// TIA Portal V20 export
FUNCTION_BLOCK "FB_IO_Device_Functional_Test"   // FB4, LAD
{ S7_Optimized_Access := 'TRUE' }
// stored: MemoryReserve 100, SetENOAutomatically false
   VAR_INPUT
      Reset_PLC_Functional_Test : Array[0..31] of Bool;
      Status : Bool;
      Voltage_Read : UInt;
      Min_Electrical_Current : UInt;
      Max_Electrical_Current : UInt;
      Time_End_Electrical_Current_Test : Time;
      Time_Start_Visual_Test : Time;
      In_Functional_Test_Odd : "IO_Device_Functinal_Test_Odd";
      In_Functional_Test_Even : "IO_Device_Functinal_Test_Even";
   END_VAR
   VAR_OUTPUT
      Out_Test_Parameters_Odd : "IO_Device_Test_Parameters_Odd";
      Out_Test_Parameters_Even : "IO_Device_Test_Parameters_Even";
      Out_Voltage_Read : UInt;
      Comunication_Error_Panel_1 : Bool;
      Comunication_Error_Panel_2 : Bool;
      Comunication_Error_Panel_3 : Bool;
      Comunication_Error_Panel_4 : Bool;
      Comunication_Error_Panel_5 : Bool;
      Comunication_Error_Panel_6 : Bool;
      Comunication_Error_Panel_7 : Bool;
      Comunication_Error_Panel_8 : Bool;
      Comunication_Error_Panel_9 : Bool;
      Comunication_Error_Panel_10 : Bool;
      Comunication_Error_Panel_11 : Bool;
      Comunication_Error_Panel_12 : Bool;
      Comunication_Error_Panel_13 : Bool;
      Comunication_Error_Panel_14 : Bool;
      Comunication_Error_Panel_15 : Bool;
      Comunication_Error_Panel_16 : Bool;
      Comunication_Error_Panel_17 : Bool;
      Comunication_Error_Panel_18 : Bool;
      Comunication_Error_Panel_19 : Bool;
      Comunication_Error_Panel_20 : Bool;
      Comunication_Error_Panel_21 : Bool;
      Comunication_Error_Panel_22 : Bool;
      Comunication_Error_Panel_23 : Bool;
      Comunication_Error_Panel_24 : Bool;
      Comunication_Error_Panel_25 : Bool;
      Comunication_Error_Panel_26 : Bool;
      Comunication_Error_Panel_27 : Bool;
      Comunication_Error_Panel_28 : Bool;
      Comunication_Error_Panel_29 : Bool;
      Comunication_Error_Panel_30 : Bool;
   END_VAR
   VAR
      Enable_Comunication_Erro_3 : Bool;
      Enable_Comunication_Erro_4 : Bool;
      Enable_Comunication_Erro_5 : Bool;
      Enable_Comunication_Erro_6 : Bool;
      Enable_Comunication_Erro_7 : Bool;
      Enable_Comunication_Erro_8 : Bool;
      Enable_Comunication_Erro_9 : Bool;
      Enable_Comunication_Erro_10 : Bool;
      Enable_Comunication_Erro_11 : Bool;
      Enable_Comunication_Erro_12 : Bool;
      Enable_Comunication_Erro_13 : Bool;
      Enable_Comunication_Erro_14 : Bool;
      Enable_Comunication_Erro_15 : Bool;
      Enable_Comunication_Erro_16 : Bool;
      Enable_Comunication_Erro_17 : Bool;
      Enable_Comunication_Erro_18 : Bool;
      Enable_Comunication_Erro_19 : Bool;
      Enable_Comunication_Erro_20 : Bool;
      Enable_Comunication_Erro_21 : Bool;
      Enable_Comunication_Erro_22 : Bool;
      Enable_Comunication_Erro_23 : Bool;
      Enable_Comunication_Erro_24 : Bool;
      Enable_Comunication_Erro_25 : Bool;
      Enable_Comunication_Erro_26 : Bool;
      Enable_Comunication_Erro_27 : Bool;
      Enable_Comunication_Erro_28 : Bool;
      Enable_Comunication_Erro_29 : Bool;
      Enable_Comunication_Erro_30 : Bool;
      Timer_Alarme_A_1 { S7_SetPoint := 'True'} : TON_TIME;
      Timer_Alarme_B_1 { S7_SetPoint := 'True'} : TON_TIME;
      Timer_Alarme_A_2 { S7_SetPoint := 'True'} : TON_TIME;
      Timer_Alarme_B_2 { S7_SetPoint := 'True'} : TON_TIME;
      Timer_Alarme_A_3 { S7_SetPoint := 'True'} : TON_TIME;
      Timer_Alarme_B_3 { S7_SetPoint := 'True'} : TON_TIME;
      Timer_Alarme_A_4 { S7_SetPoint := 'True'} : TON_TIME;
      Timer_Alarme_B_4 { S7_SetPoint := 'True'} : TON_TIME;
      Timer_Alarme_A_5 { S7_SetPoint := 'True'} : TON_TIME;
      Timer_Alarme_B_5 { S7_SetPoint := 'True'} : TON_TIME;
      Timer_Alarme_A_6 { S7_SetPoint := 'True'} : TON_TIME;
      Timer_Alarme_B_6 { S7_SetPoint := 'True'} : TON_TIME;
      Timer_Alarme_A_7 { S7_SetPoint := 'True'} : TON_TIME;
      Timer_Alarme_B_7 { S7_SetPoint := 'True'} : TON_TIME;
      Timer_Alarme_A_8 { S7_SetPoint := 'True'} : TON_TIME;
      Timer_Alarme_B_8 { S7_SetPoint := 'True'} : TON_TIME;
      Timer_Alarme_A_9 { S7_SetPoint := 'True'} : TON_TIME;
      Timer_Alarme_B_9 { S7_SetPoint := 'True'} : TON_TIME;
      Timer_Alarme_A_10 { S7_SetPoint := 'True'} : TON_TIME;
      Timer_Alarme_B_10 { S7_SetPoint := 'True'} : TON_TIME;
      Timer_Alarme_A_11 { S7_SetPoint := 'True'} : TON_TIME;
      Timer_Alarme_B_11 { S7_SetPoint := 'True'} : TON_TIME;
      Timer_Alarme_A_12 { S7_SetPoint := 'True'} : TON_TIME;
      Timer_Alarme_B_12 { S7_SetPoint := 'True'} : TON_TIME;
      Timer_Alarme_A_13 { S7_SetPoint := 'True'} : TON_TIME;
      Timer_Alarme_B_13 { S7_SetPoint := 'True'} : TON_TIME;
      Timer_Alarme_A_14 { S7_SetPoint := 'True'} : TON_TIME;
      Timer_Alarme_B_14 { S7_SetPoint := 'True'} : TON_TIME;
      Timer_Alarme_A_15 { S7_SetPoint := 'True'} : TON_TIME;
      Timer_Alarme_B_15 { S7_SetPoint := 'True'} : TON_TIME;
      Timer_Alarme_A_16 { S7_SetPoint := 'True'} : TON_TIME;
      Timer_Alarme_B_16 { S7_SetPoint := 'True'} : TON_TIME;
      Timer_Alarme_A_17 { S7_SetPoint := 'True'} : TON_TIME;
      Timer_Alarme_B_17 { S7_SetPoint := 'True'} : TON_TIME;
      Timer_Alarme_A_18 { S7_SetPoint := 'True'} : TON_TIME;
      Timer_Alarme_B_18 { S7_SetPoint := 'True'} : TON_TIME;
      Timer_Alarme_A_19 { S7_SetPoint := 'True'} : TON_TIME;
      Timer_Alarme_B_19 { S7_SetPoint := 'True'} : TON_TIME;
      Timer_Alarme_A_20 { S7_SetPoint := 'True'} : TON_TIME;
      Timer_Alarme_B_20 { S7_SetPoint := 'True'} : TON_TIME;
      Timer_Alarme_A_21 { S7_SetPoint := 'True'} : TON_TIME;
      Timer_Alarme_B_21 { S7_SetPoint := 'True'} : TON_TIME;
      Timer_Alarme_A_22 { S7_SetPoint := 'True'} : TON_TIME;
      Timer_Alarme_B_22 { S7_SetPoint := 'True'} : TON_TIME;
      Timer_Alarme_A_23 { S7_SetPoint := 'True'} : TON_TIME;
      Timer_Alarme_B_23 { S7_SetPoint := 'True'} : TON_TIME;
      Timer_Alarme_A_24 { S7_SetPoint := 'True'} : TON_TIME;
      Timer_Alarme_B_24 { S7_SetPoint := 'True'} : TON_TIME;
      Timer_Alarme_A_25 { S7_SetPoint := 'True'} : TON_TIME;
      Timer_Alarme_B_25 { S7_SetPoint := 'True'} : TON_TIME;
      Timer_Alarme_A_26 { S7_SetPoint := 'True'} : TON_TIME;
      Timer_Alarme_B_26 { S7_SetPoint := 'True'} : TON_TIME;
      Timer_Alarme_A_27 { S7_SetPoint := 'True'} : TON_TIME;
      Timer_Alarme_B_27 { S7_SetPoint := 'True'} : TON_TIME;
      Timer_Alarme_A_28 { S7_SetPoint := 'True'} : TON_TIME;
      Timer_Alarme_B_28 { S7_SetPoint := 'True'} : TON_TIME;
      Timer_Alarme_A_29 { S7_SetPoint := 'True'} : TON_TIME;
      Timer_Alarme_B_29 { S7_SetPoint := 'True'} : TON_TIME;
      Timer_Alarme_A_30 { S7_SetPoint := 'True'} : TON_TIME;
      Timer_Alarme_B_30 { S7_SetPoint := 'True'} : TON_TIME;
   END_VAR
BEGIN

REGION Network 1
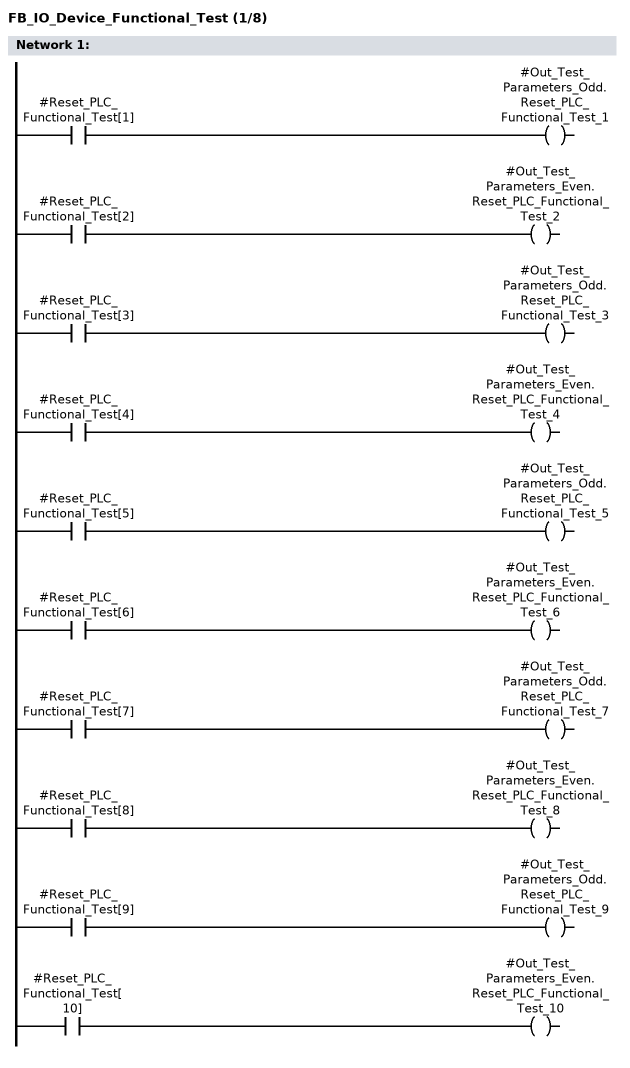
   RUNG wire#powerrail
      Contact( #Reset_PLC_Functional_Test[1] )
      Coil( #Out_Test_Parameters_Odd.Reset_PLC_Functional_Test_1 )
   END_RUNG
   RUNG wire#powerrail
      Contact( #Reset_PLC_Functional_Test[2] )
      Coil( #Out_Test_Parameters_Even.Reset_PLC_Functional_Test_2 )
   END_RUNG
   RUNG wire#powerrail
      Contact( #Reset_PLC_Functional_Test[3] )
      Coil( #Out_Test_Parameters_Odd.Reset_PLC_Functional_Test_3 )
   END_RUNG
   RUNG wire#powerrail
      Contact( #Reset_PLC_Functional_Test[4] )
      Coil( #Out_Test_Parameters_Even.Reset_PLC_Functional_Test_4 )
   END_RUNG
   RUNG wire#powerrail
      Contact( #Reset_PLC_Functional_Test[5] )
      Coil( #Out_Test_Parameters_Odd.Reset_PLC_Functional_Test_5 )
   END_RUNG
   RUNG wire#powerrail
      Contact( #Reset_PLC_Functional_Test[6] )
      Coil( #Out_Test_Parameters_Even.Reset_PLC_Functional_Test_6 )
   END_RUNG
   RUNG wire#powerrail
      Contact( #Reset_PLC_Functional_Test[7] )
      Coil( #Out_Test_Parameters_Odd.Reset_PLC_Functional_Test_7 )
   END_RUNG
   RUNG wire#powerrail
      Contact( #Reset_PLC_Functional_Test[8] )
      Coil( #Out_Test_Parameters_Even.Reset_PLC_Functional_Test_8 )
   END_RUNG
   RUNG wire#powerrail
      Contact( #Reset_PLC_Functional_Test[9] )
      Coil( #Out_Test_Parameters_Odd.Reset_PLC_Functional_Test_9 )
   END_RUNG
   RUNG wire#powerrail
      Contact( #Reset_PLC_Functional_Test[10] )
      Coil( #Out_Test_Parameters_Even.Reset_PLC_Functional_Test_10 )
   END_RUNG
   // the same network as SCL:
   #Out_Test_Parameters_Odd.Reset_PLC_Functional_Test_1 := #Reset_PLC_Functional_Test[1];
   #Out_Test_Parameters_Even.Reset_PLC_Functional_Test_2 := #Reset_PLC_Functional_Test[2];
   #Out_Test_Parameters_Odd.Reset_PLC_Functional_Test_3 := #Reset_PLC_Functional_Test[3];
   #Out_Test_Parameters_Even.Reset_PLC_Functional_Test_4 := #Reset_PLC_Functional_Test[4];
   #Out_Test_Parameters_Odd.Reset_PLC_Functional_Test_5 := #Reset_PLC_Functional_Test[5];
   #Out_Test_Parameters_Even.Reset_PLC_Functional_Test_6 := #Reset_PLC_Functional_Test[6];
   #Out_Test_Parameters_Odd.Reset_PLC_Functional_Test_7 := #Reset_PLC_Functional_Test[7];
   #Out_Test_Parameters_Even.Reset_PLC_Functional_Test_8 := #Reset_PLC_Functional_Test[8];
   #Out_Test_Parameters_Odd.Reset_PLC_Functional_Test_9 := #Reset_PLC_Functional_Test[9];
   #Out_Test_Parameters_Even.Reset_PLC_Functional_Test_10 := #Reset_PLC_Functional_Test[10];
END_REGION

REGION Network 2
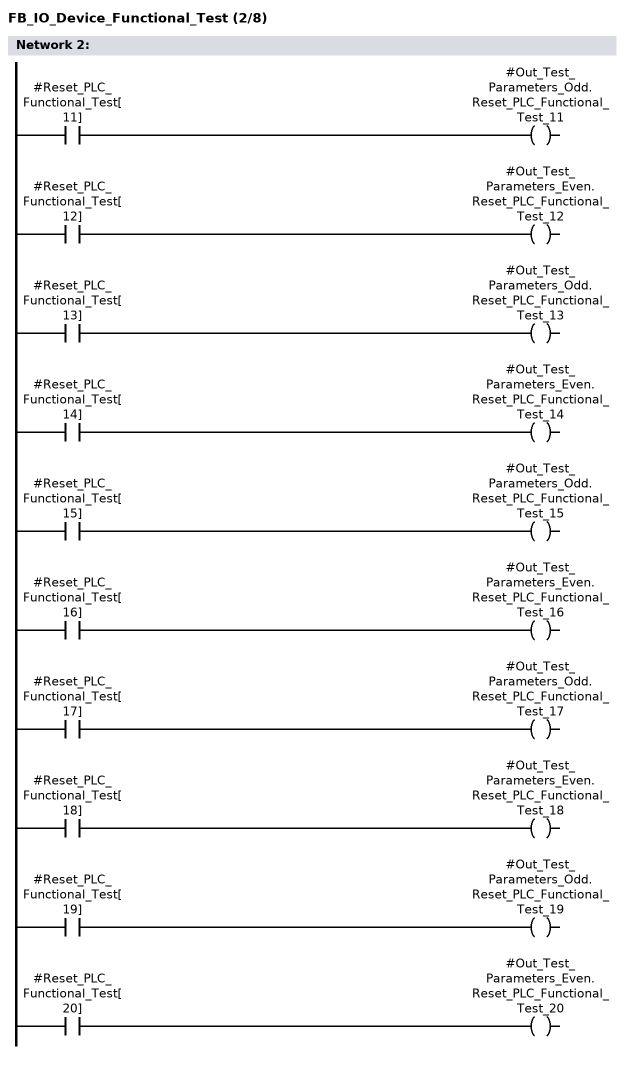
   RUNG wire#powerrail
      Contact( #Reset_PLC_Functional_Test[11] )
      Coil( #Out_Test_Parameters_Odd.Reset_PLC_Functional_Test_11 )
   END_RUNG
   RUNG wire#powerrail
      Contact( #Reset_PLC_Functional_Test[12] )
      Coil( #Out_Test_Parameters_Even.Reset_PLC_Functional_Test_12 )
   END_RUNG
   RUNG wire#powerrail
      Contact( #Reset_PLC_Functional_Test[13] )
      Coil( #Out_Test_Parameters_Odd.Reset_PLC_Functional_Test_13 )
   END_RUNG
   RUNG wire#powerrail
      Contact( #Reset_PLC_Functional_Test[14] )
      Coil( #Out_Test_Parameters_Even.Reset_PLC_Functional_Test_14 )
   END_RUNG
   RUNG wire#powerrail
      Contact( #Reset_PLC_Functional_Test[15] )
      Coil( #Out_Test_Parameters_Odd.Reset_PLC_Functional_Test_15 )
   END_RUNG
   RUNG wire#powerrail
      Contact( #Reset_PLC_Functional_Test[16] )
      Coil( #Out_Test_Parameters_Even.Reset_PLC_Functional_Test_16 )
   END_RUNG
   RUNG wire#powerrail
      Contact( #Reset_PLC_Functional_Test[17] )
      Coil( #Out_Test_Parameters_Odd.Reset_PLC_Functional_Test_17 )
   END_RUNG
   RUNG wire#powerrail
      Contact( #Reset_PLC_Functional_Test[18] )
      Coil( #Out_Test_Parameters_Even.Reset_PLC_Functional_Test_18 )
   END_RUNG
   RUNG wire#powerrail
      Contact( #Reset_PLC_Functional_Test[19] )
      Coil( #Out_Test_Parameters_Odd.Reset_PLC_Functional_Test_19 )
   END_RUNG
   RUNG wire#powerrail
      Contact( #Reset_PLC_Functional_Test[20] )
      Coil( #Out_Test_Parameters_Even.Reset_PLC_Functional_Test_20 )
   END_RUNG
   // the same network as SCL:
   #Out_Test_Parameters_Odd.Reset_PLC_Functional_Test_11 := #Reset_PLC_Functional_Test[11];
   #Out_Test_Parameters_Even.Reset_PLC_Functional_Test_12 := #Reset_PLC_Functional_Test[12];
   #Out_Test_Parameters_Odd.Reset_PLC_Functional_Test_13 := #Reset_PLC_Functional_Test[13];
   #Out_Test_Parameters_Even.Reset_PLC_Functional_Test_14 := #Reset_PLC_Functional_Test[14];
   #Out_Test_Parameters_Odd.Reset_PLC_Functional_Test_15 := #Reset_PLC_Functional_Test[15];
   #Out_Test_Parameters_Even.Reset_PLC_Functional_Test_16 := #Reset_PLC_Functional_Test[16];
   #Out_Test_Parameters_Odd.Reset_PLC_Functional_Test_17 := #Reset_PLC_Functional_Test[17];
   #Out_Test_Parameters_Even.Reset_PLC_Functional_Test_18 := #Reset_PLC_Functional_Test[18];
   #Out_Test_Parameters_Odd.Reset_PLC_Functional_Test_19 := #Reset_PLC_Functional_Test[19];
   #Out_Test_Parameters_Even.Reset_PLC_Functional_Test_20 := #Reset_PLC_Functional_Test[20];
END_REGION

REGION Network 3
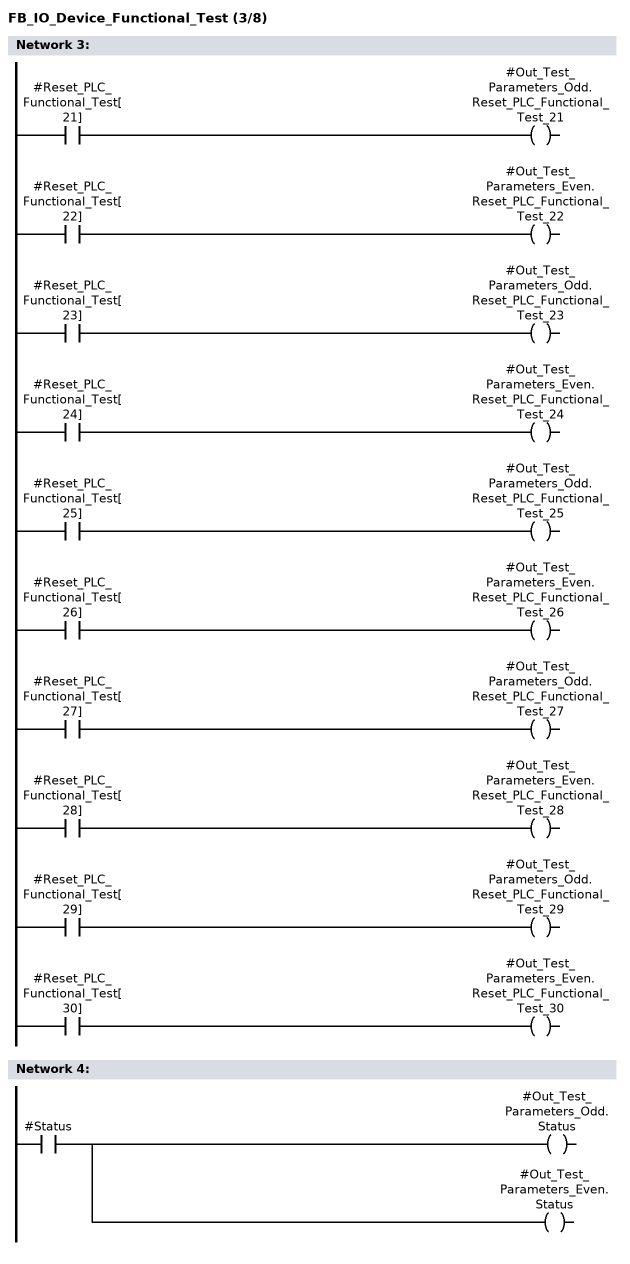
   RUNG wire#powerrail
      Contact( #Reset_PLC_Functional_Test[21] )
      Coil( #Out_Test_Parameters_Odd.Reset_PLC_Functional_Test_21 )
   END_RUNG
   RUNG wire#powerrail
      Contact( #Reset_PLC_Functional_Test[22] )
      Coil( #Out_Test_Parameters_Even.Reset_PLC_Functional_Test_22 )
   END_RUNG
   RUNG wire#powerrail
      Contact( #Reset_PLC_Functional_Test[23] )
      Coil( #Out_Test_Parameters_Odd.Reset_PLC_Functional_Test_23 )
   END_RUNG
   RUNG wire#powerrail
      Contact( #Reset_PLC_Functional_Test[24] )
      Coil( #Out_Test_Parameters_Even.Reset_PLC_Functional_Test_24 )
   END_RUNG
   RUNG wire#powerrail
      Contact( #Reset_PLC_Functional_Test[25] )
      Coil( #Out_Test_Parameters_Odd.Reset_PLC_Functional_Test_25 )
   END_RUNG
   RUNG wire#powerrail
      Contact( #Reset_PLC_Functional_Test[26] )
      Coil( #Out_Test_Parameters_Even.Reset_PLC_Functional_Test_26 )
   END_RUNG
   RUNG wire#powerrail
      Contact( #Reset_PLC_Functional_Test[27] )
      Coil( #Out_Test_Parameters_Odd.Reset_PLC_Functional_Test_27 )
   END_RUNG
   RUNG wire#powerrail
      Contact( #Reset_PLC_Functional_Test[28] )
      Coil( #Out_Test_Parameters_Even.Reset_PLC_Functional_Test_28 )
   END_RUNG
   RUNG wire#powerrail
      Contact( #Reset_PLC_Functional_Test[29] )
      Coil( #Out_Test_Parameters_Odd.Reset_PLC_Functional_Test_29 )
   END_RUNG
   RUNG wire#powerrail
      Contact( #Reset_PLC_Functional_Test[30] )
      Coil( #Out_Test_Parameters_Even.Reset_PLC_Functional_Test_30 )
   END_RUNG
   // the same network as SCL:
   #Out_Test_Parameters_Odd.Reset_PLC_Functional_Test_21 := #Reset_PLC_Functional_Test[21];
   #Out_Test_Parameters_Even.Reset_PLC_Functional_Test_22 := #Reset_PLC_Functional_Test[22];
   #Out_Test_Parameters_Odd.Reset_PLC_Functional_Test_23 := #Reset_PLC_Functional_Test[23];
   #Out_Test_Parameters_Even.Reset_PLC_Functional_Test_24 := #Reset_PLC_Functional_Test[24];
   #Out_Test_Parameters_Odd.Reset_PLC_Functional_Test_25 := #Reset_PLC_Functional_Test[25];
   #Out_Test_Parameters_Even.Reset_PLC_Functional_Test_26 := #Reset_PLC_Functional_Test[26];
   #Out_Test_Parameters_Odd.Reset_PLC_Functional_Test_27 := #Reset_PLC_Functional_Test[27];
   #Out_Test_Parameters_Even.Reset_PLC_Functional_Test_28 := #Reset_PLC_Functional_Test[28];
   #Out_Test_Parameters_Odd.Reset_PLC_Functional_Test_29 := #Reset_PLC_Functional_Test[29];
   #Out_Test_Parameters_Even.Reset_PLC_Functional_Test_30 := #Reset_PLC_Functional_Test[30];
END_REGION

REGION Network 4
   RUNG wire#powerrail
      Contact( #Status )
      wire#w1
      Coil( #Out_Test_Parameters_Odd.Status )
   END_RUNG
   RUNG wire#w1
      Coil( #Out_Test_Parameters_Even.Status )
   END_RUNG
   // the same network as SCL:
   #Out_Test_Parameters_Odd.Status := #Status;
   #Out_Test_Parameters_Even.Status := #Status;
END_REGION

REGION Network 5
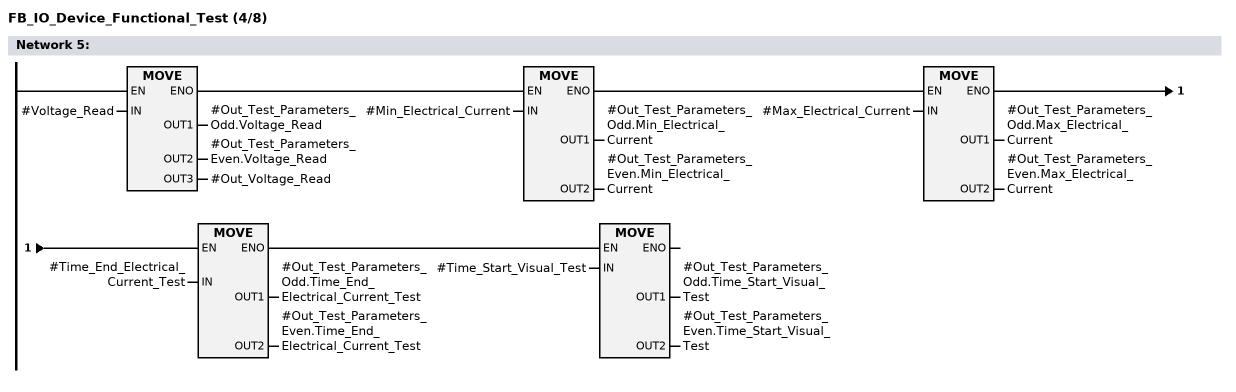
   RUNG wire#powerrail
      Move(in := #Voltage_Read, out1 => #Out_Test_Parameters_Odd.Voltage_Read, out2 => #Out_Test_Parameters_Even.Voltage_Read, out3 => #Out_Voltage_Read)
      Move(in := #Min_Electrical_Current, out1 => #Out_Test_Parameters_Odd.Min_Electrical_Current, out2 => #Out_Test_Parameters_Even.Min_Electrical_Current)
      Move(in := #Max_Electrical_Current, out1 => #Out_Test_Parameters_Odd.Max_Electrical_Current, out2 => #Out_Test_Parameters_Even.Max_Electrical_Current)
      Move(in := #Time_End_Electrical_Current_Test, out1 => #Out_Test_Parameters_Odd.Time_End_Electrical_Current_Test, out2 => #Out_Test_Parameters_Even.Time_End_Electrical_Current_Test)
      Move(in := #Time_Start_Visual_Test, out1 => #Out_Test_Parameters_Odd.Time_Start_Visual_Test, out2 => #Out_Test_Parameters_Even.Time_Start_Visual_Test)
   END_RUNG
   // the same network as SCL:
   #Out_Test_Parameters_Odd.Voltage_Read := #Voltage_Read;
   #Out_Test_Parameters_Even.Voltage_Read := #Voltage_Read;
   #Out_Voltage_Read := #Voltage_Read;
   #Out_Test_Parameters_Odd.Min_Electrical_Current := #Min_Electrical_Current;
   #Out_Test_Parameters_Even.Min_Electrical_Current := #Min_Electrical_Current;
   #Out_Test_Parameters_Odd.Max_Electrical_Current := #Max_Electrical_Current;
   #Out_Test_Parameters_Even.Max_Electrical_Current := #Max_Electrical_Current;
   #Out_Test_Parameters_Odd.Time_End_Electrical_Current_Test := #Time_End_Electrical_Current_Test;
   #Out_Test_Parameters_Even.Time_End_Electrical_Current_Test := #Time_End_Electrical_Current_Test;
   #Out_Test_Parameters_Odd.Time_Start_Visual_Test := #Time_Start_Visual_Test;
   #Out_Test_Parameters_Even.Time_Start_Visual_Test := #Time_Start_Visual_Test;
END_REGION

REGION Network 6
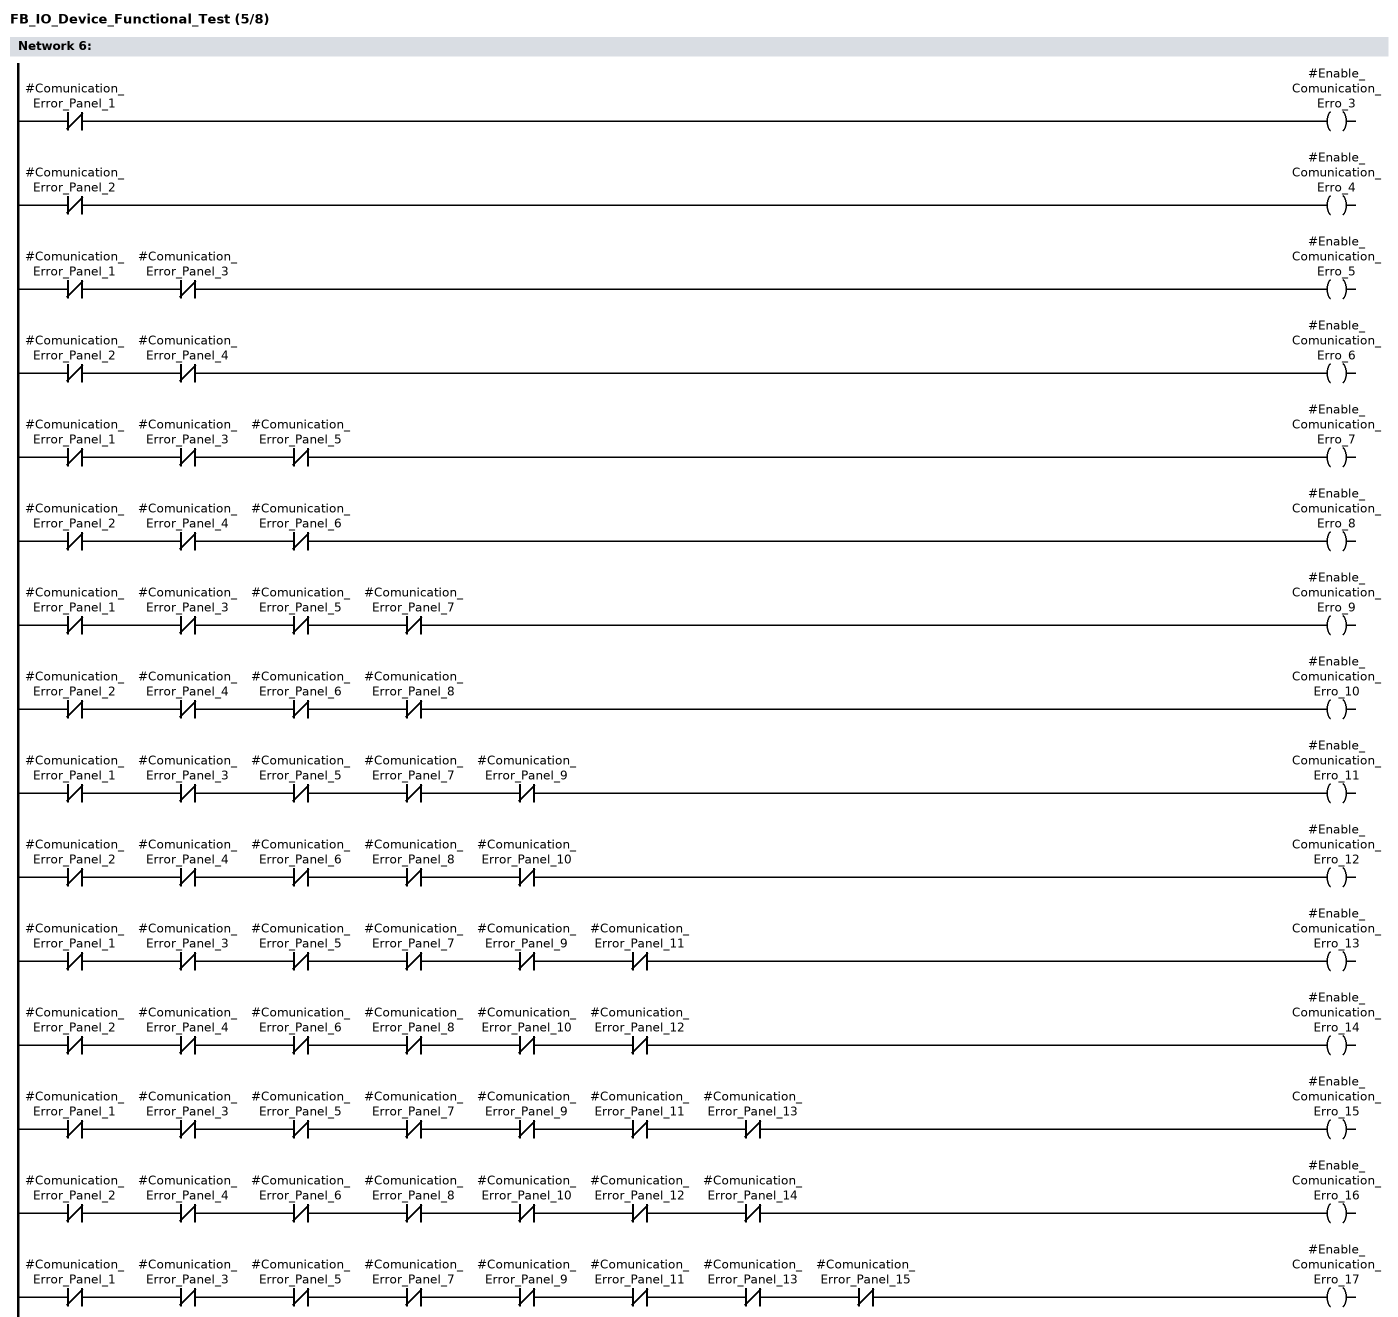
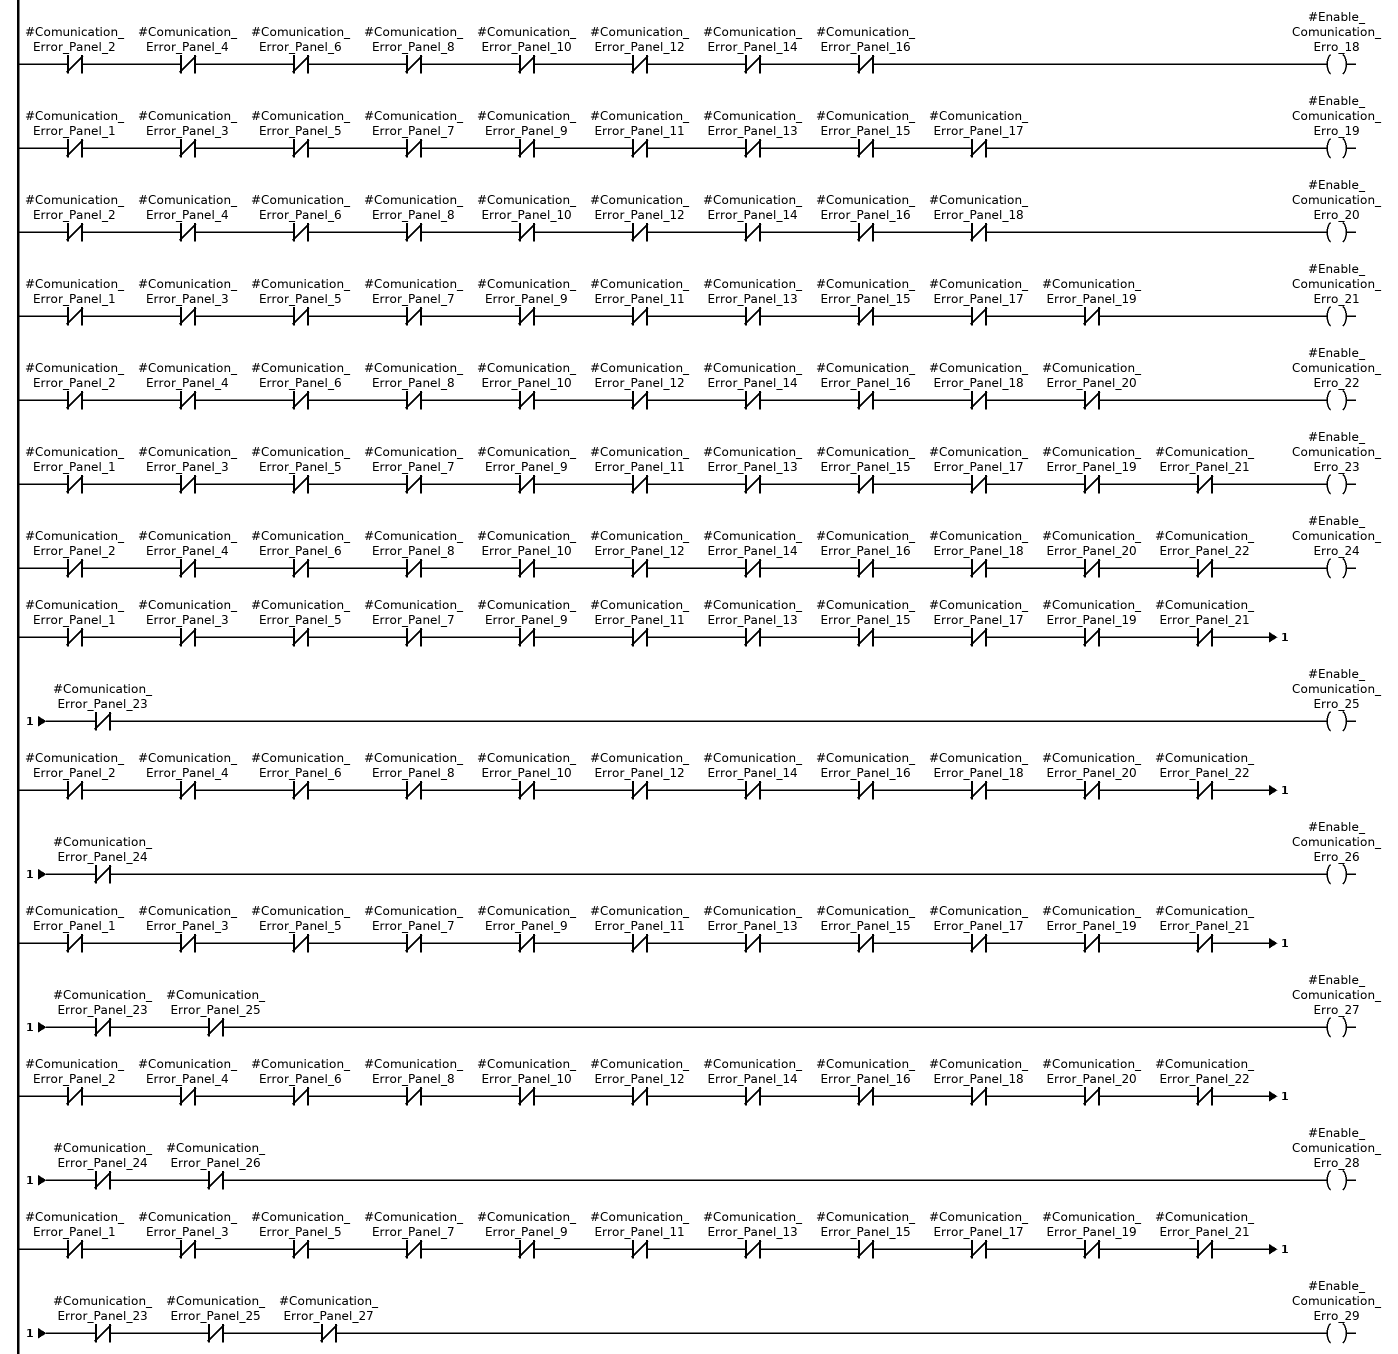
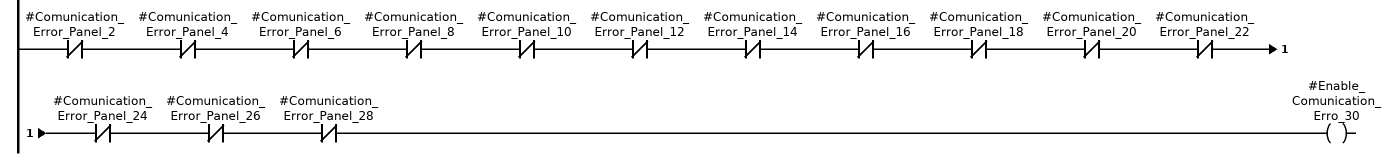
   RUNG wire#powerrail
      I_Contact( #Comunication_Error_Panel_1 )
      Coil( #Enable_Comunication_Erro_3 )
   END_RUNG
   RUNG wire#powerrail
      I_Contact( #Comunication_Error_Panel_2 )
      Coil( #Enable_Comunication_Erro_4 )
   END_RUNG
   RUNG wire#powerrail
      I_Contact( #Comunication_Error_Panel_1 )
      I_Contact( #Comunication_Error_Panel_3 )
      Coil( #Enable_Comunication_Erro_5 )
   END_RUNG
   RUNG wire#powerrail
      I_Contact( #Comunication_Error_Panel_2 )
      I_Contact( #Comunication_Error_Panel_4 )
      Coil( #Enable_Comunication_Erro_6 )
   END_RUNG
   RUNG wire#powerrail
      I_Contact( #Comunication_Error_Panel_1 )
      I_Contact( #Comunication_Error_Panel_3 )
      I_Contact( #Comunication_Error_Panel_5 )
      Coil( #Enable_Comunication_Erro_7 )
   END_RUNG
   RUNG wire#powerrail
      I_Contact( #Comunication_Error_Panel_2 )
      I_Contact( #Comunication_Error_Panel_4 )
      I_Contact( #Comunication_Error_Panel_6 )
      Coil( #Enable_Comunication_Erro_8 )
   END_RUNG
   RUNG wire#powerrail
      I_Contact( #Comunication_Error_Panel_1 )
      I_Contact( #Comunication_Error_Panel_3 )
      I_Contact( #Comunication_Error_Panel_5 )
      I_Contact( #Comunication_Error_Panel_7 )
      Coil( #Enable_Comunication_Erro_9 )
   END_RUNG
   RUNG wire#powerrail
      I_Contact( #Comunication_Error_Panel_2 )
      I_Contact( #Comunication_Error_Panel_4 )
      I_Contact( #Comunication_Error_Panel_6 )
      I_Contact( #Comunication_Error_Panel_8 )
      Coil( #Enable_Comunication_Erro_10 )
   END_RUNG
   RUNG wire#powerrail
      I_Contact( #Comunication_Error_Panel_1 )
      I_Contact( #Comunication_Error_Panel_3 )
      I_Contact( #Comunication_Error_Panel_5 )
      I_Contact( #Comunication_Error_Panel_7 )
      I_Contact( #Comunication_Error_Panel_9 )
      Coil( #Enable_Comunication_Erro_11 )
   END_RUNG
   RUNG wire#powerrail
      I_Contact( #Comunication_Error_Panel_2 )
      I_Contact( #Comunication_Error_Panel_4 )
      I_Contact( #Comunication_Error_Panel_6 )
      I_Contact( #Comunication_Error_Panel_8 )
      I_Contact( #Comunication_Error_Panel_10 )
      Coil( #Enable_Comunication_Erro_12 )
   END_RUNG
   RUNG wire#powerrail
      I_Contact( #Comunication_Error_Panel_1 )
      I_Contact( #Comunication_Error_Panel_3 )
      I_Contact( #Comunication_Error_Panel_5 )
      I_Contact( #Comunication_Error_Panel_7 )
      I_Contact( #Comunication_Error_Panel_9 )
      I_Contact( #Comunication_Error_Panel_11 )
      Coil( #Enable_Comunication_Erro_13 )
   END_RUNG
   RUNG wire#powerrail
      I_Contact( #Comunication_Error_Panel_2 )
      I_Contact( #Comunication_Error_Panel_4 )
      I_Contact( #Comunication_Error_Panel_6 )
      I_Contact( #Comunication_Error_Panel_8 )
      I_Contact( #Comunication_Error_Panel_10 )
      I_Contact( #Comunication_Error_Panel_12 )
      Coil( #Enable_Comunication_Erro_14 )
   END_RUNG
   RUNG wire#powerrail
      I_Contact( #Comunication_Error_Panel_1 )
      I_Contact( #Comunication_Error_Panel_3 )
      I_Contact( #Comunication_Error_Panel_5 )
      I_Contact( #Comunication_Error_Panel_7 )
      I_Contact( #Comunication_Error_Panel_9 )
      I_Contact( #Comunication_Error_Panel_11 )
      I_Contact( #Comunication_Error_Panel_13 )
      Coil( #Enable_Comunication_Erro_15 )
   END_RUNG
   RUNG wire#powerrail
      I_Contact( #Comunication_Error_Panel_2 )
      I_Contact( #Comunication_Error_Panel_4 )
      I_Contact( #Comunication_Error_Panel_6 )
      I_Contact( #Comunication_Error_Panel_8 )
      I_Contact( #Comunication_Error_Panel_10 )
      I_Contact( #Comunication_Error_Panel_12 )
      I_Contact( #Comunication_Error_Panel_14 )
      Coil( #Enable_Comunication_Erro_16 )
   END_RUNG
   RUNG wire#powerrail
      I_Contact( #Comunication_Error_Panel_1 )
      I_Contact( #Comunication_Error_Panel_3 )
      I_Contact( #Comunication_Error_Panel_5 )
      I_Contact( #Comunication_Error_Panel_7 )
      I_Contact( #Comunication_Error_Panel_9 )
      I_Contact( #Comunication_Error_Panel_11 )
      I_Contact( #Comunication_Error_Panel_13 )
      I_Contact( #Comunication_Error_Panel_15 )
      Coil( #Enable_Comunication_Erro_17 )
   END_RUNG
   RUNG wire#powerrail
      I_Contact( #Comunication_Error_Panel_2 )
      I_Contact( #Comunication_Error_Panel_4 )
      I_Contact( #Comunication_Error_Panel_6 )
      I_Contact( #Comunication_Error_Panel_8 )
      I_Contact( #Comunication_Error_Panel_10 )
      I_Contact( #Comunication_Error_Panel_12 )
      I_Contact( #Comunication_Error_Panel_14 )
      I_Contact( #Comunication_Error_Panel_16 )
      Coil( #Enable_Comunication_Erro_18 )
   END_RUNG
   RUNG wire#powerrail
      I_Contact( #Comunication_Error_Panel_1 )
      I_Contact( #Comunication_Error_Panel_3 )
      I_Contact( #Comunication_Error_Panel_5 )
      I_Contact( #Comunication_Error_Panel_7 )
      I_Contact( #Comunication_Error_Panel_9 )
      I_Contact( #Comunication_Error_Panel_11 )
      I_Contact( #Comunication_Error_Panel_13 )
      I_Contact( #Comunication_Error_Panel_15 )
      I_Contact( #Comunication_Error_Panel_17 )
      Coil( #Enable_Comunication_Erro_19 )
   END_RUNG
   RUNG wire#powerrail
      I_Contact( #Comunication_Error_Panel_2 )
      I_Contact( #Comunication_Error_Panel_4 )
      I_Contact( #Comunication_Error_Panel_6 )
      I_Contact( #Comunication_Error_Panel_8 )
      I_Contact( #Comunication_Error_Panel_10 )
      I_Contact( #Comunication_Error_Panel_12 )
      I_Contact( #Comunication_Error_Panel_14 )
      I_Contact( #Comunication_Error_Panel_16 )
      I_Contact( #Comunication_Error_Panel_18 )
      Coil( #Enable_Comunication_Erro_20 )
   END_RUNG
   RUNG wire#powerrail
      I_Contact( #Comunication_Error_Panel_1 )
      I_Contact( #Comunication_Error_Panel_3 )
      I_Contact( #Comunication_Error_Panel_5 )
      I_Contact( #Comunication_Error_Panel_7 )
      I_Contact( #Comunication_Error_Panel_9 )
      I_Contact( #Comunication_Error_Panel_11 )
      I_Contact( #Comunication_Error_Panel_13 )
      I_Contact( #Comunication_Error_Panel_15 )
      I_Contact( #Comunication_Error_Panel_17 )
      I_Contact( #Comunication_Error_Panel_19 )
      Coil( #Enable_Comunication_Erro_21 )
   END_RUNG
   RUNG wire#powerrail
      I_Contact( #Comunication_Error_Panel_2 )
      I_Contact( #Comunication_Error_Panel_4 )
      I_Contact( #Comunication_Error_Panel_6 )
      I_Contact( #Comunication_Error_Panel_8 )
      I_Contact( #Comunication_Error_Panel_10 )
      I_Contact( #Comunication_Error_Panel_12 )
      I_Contact( #Comunication_Error_Panel_14 )
      I_Contact( #Comunication_Error_Panel_16 )
      I_Contact( #Comunication_Error_Panel_18 )
      I_Contact( #Comunication_Error_Panel_20 )
      Coil( #Enable_Comunication_Erro_22 )
   END_RUNG
   RUNG wire#powerrail
      I_Contact( #Comunication_Error_Panel_1 )
      I_Contact( #Comunication_Error_Panel_3 )
      I_Contact( #Comunication_Error_Panel_5 )
      I_Contact( #Comunication_Error_Panel_7 )
      I_Contact( #Comunication_Error_Panel_9 )
      I_Contact( #Comunication_Error_Panel_11 )
      I_Contact( #Comunication_Error_Panel_13 )
      I_Contact( #Comunication_Error_Panel_15 )
      I_Contact( #Comunication_Error_Panel_17 )
      I_Contact( #Comunication_Error_Panel_19 )
      I_Contact( #Comunication_Error_Panel_21 )
      Coil( #Enable_Comunication_Erro_23 )
   END_RUNG
   RUNG wire#powerrail
      I_Contact( #Comunication_Error_Panel_2 )
      I_Contact( #Comunication_Error_Panel_4 )
      I_Contact( #Comunication_Error_Panel_6 )
      I_Contact( #Comunication_Error_Panel_8 )
      I_Contact( #Comunication_Error_Panel_10 )
      I_Contact( #Comunication_Error_Panel_12 )
      I_Contact( #Comunication_Error_Panel_14 )
      I_Contact( #Comunication_Error_Panel_16 )
      I_Contact( #Comunication_Error_Panel_18 )
      I_Contact( #Comunication_Error_Panel_20 )
      I_Contact( #Comunication_Error_Panel_22 )
      Coil( #Enable_Comunication_Erro_24 )
   END_RUNG
   RUNG wire#powerrail
      I_Contact( #Comunication_Error_Panel_1 )
      I_Contact( #Comunication_Error_Panel_3 )
      I_Contact( #Comunication_Error_Panel_5 )
      I_Contact( #Comunication_Error_Panel_7 )
      I_Contact( #Comunication_Error_Panel_9 )
      I_Contact( #Comunication_Error_Panel_11 )
      I_Contact( #Comunication_Error_Panel_13 )
      I_Contact( #Comunication_Error_Panel_15 )
      I_Contact( #Comunication_Error_Panel_17 )
      I_Contact( #Comunication_Error_Panel_19 )
      I_Contact( #Comunication_Error_Panel_21 )
      I_Contact( #Comunication_Error_Panel_23 )
      Coil( #Enable_Comunication_Erro_25 )
   END_RUNG
   RUNG wire#powerrail
      I_Contact( #Comunication_Error_Panel_2 )
      I_Contact( #Comunication_Error_Panel_4 )
      I_Contact( #Comunication_Error_Panel_6 )
      I_Contact( #Comunication_Error_Panel_8 )
      I_Contact( #Comunication_Error_Panel_10 )
      I_Contact( #Comunication_Error_Panel_12 )
      I_Contact( #Comunication_Error_Panel_14 )
      I_Contact( #Comunication_Error_Panel_16 )
      I_Contact( #Comunication_Error_Panel_18 )
      I_Contact( #Comunication_Error_Panel_20 )
      I_Contact( #Comunication_Error_Panel_22 )
      I_Contact( #Comunication_Error_Panel_24 )
      Coil( #Enable_Comunication_Erro_26 )
   END_RUNG
   RUNG wire#powerrail
      I_Contact( #Comunication_Error_Panel_1 )
      I_Contact( #Comunication_Error_Panel_3 )
      I_Contact( #Comunication_Error_Panel_5 )
      I_Contact( #Comunication_Error_Panel_7 )
      I_Contact( #Comunication_Error_Panel_9 )
      I_Contact( #Comunication_Error_Panel_11 )
      I_Contact( #Comunication_Error_Panel_13 )
      I_Contact( #Comunication_Error_Panel_15 )
      I_Contact( #Comunication_Error_Panel_17 )
      I_Contact( #Comunication_Error_Panel_19 )
      I_Contact( #Comunication_Error_Panel_21 )
      I_Contact( #Comunication_Error_Panel_23 )
      I_Contact( #Comunication_Error_Panel_25 )
      Coil( #Enable_Comunication_Erro_27 )
   END_RUNG
   RUNG wire#powerrail
      I_Contact( #Comunication_Error_Panel_2 )
      I_Contact( #Comunication_Error_Panel_4 )
      I_Contact( #Comunication_Error_Panel_6 )
      I_Contact( #Comunication_Error_Panel_8 )
      I_Contact( #Comunication_Error_Panel_10 )
      I_Contact( #Comunication_Error_Panel_12 )
      I_Contact( #Comunication_Error_Panel_14 )
      I_Contact( #Comunication_Error_Panel_16 )
      I_Contact( #Comunication_Error_Panel_18 )
      I_Contact( #Comunication_Error_Panel_20 )
      I_Contact( #Comunication_Error_Panel_22 )
      I_Contact( #Comunication_Error_Panel_24 )
      I_Contact( #Comunication_Error_Panel_26 )
      Coil( #Enable_Comunication_Erro_28 )
   END_RUNG
   RUNG wire#powerrail
      I_Contact( #Comunication_Error_Panel_1 )
      I_Contact( #Comunication_Error_Panel_3 )
      I_Contact( #Comunication_Error_Panel_5 )
      I_Contact( #Comunication_Error_Panel_7 )
      I_Contact( #Comunication_Error_Panel_9 )
      I_Contact( #Comunication_Error_Panel_11 )
      I_Contact( #Comunication_Error_Panel_13 )
      I_Contact( #Comunication_Error_Panel_15 )
      I_Contact( #Comunication_Error_Panel_17 )
      I_Contact( #Comunication_Error_Panel_19 )
      I_Contact( #Comunication_Error_Panel_21 )
      I_Contact( #Comunication_Error_Panel_23 )
      I_Contact( #Comunication_Error_Panel_25 )
      I_Contact( #Comunication_Error_Panel_27 )
      Coil( #Enable_Comunication_Erro_29 )
   END_RUNG
   RUNG wire#powerrail
      I_Contact( #Comunication_Error_Panel_2 )
      I_Contact( #Comunication_Error_Panel_4 )
      I_Contact( #Comunication_Error_Panel_6 )
      I_Contact( #Comunication_Error_Panel_8 )
      I_Contact( #Comunication_Error_Panel_10 )
      I_Contact( #Comunication_Error_Panel_12 )
      I_Contact( #Comunication_Error_Panel_14 )
      I_Contact( #Comunication_Error_Panel_16 )
      I_Contact( #Comunication_Error_Panel_18 )
      I_Contact( #Comunication_Error_Panel_20 )
      I_Contact( #Comunication_Error_Panel_22 )
      I_Contact( #Comunication_Error_Panel_24 )
      I_Contact( #Comunication_Error_Panel_26 )
      I_Contact( #Comunication_Error_Panel_28 )
      Coil( #Enable_Comunication_Erro_30 )
   END_RUNG
   // the same network as SCL:
   #Enable_Comunication_Erro_3 := NOT #Comunication_Error_Panel_1;
   #Enable_Comunication_Erro_4 := NOT #Comunication_Error_Panel_2;
   #Enable_Comunication_Erro_5 := NOT #Comunication_Error_Panel_1 AND NOT #Comunication_Error_Panel_3;
   #Enable_Comunication_Erro_6 := NOT #Comunication_Error_Panel_2 AND NOT #Comunication_Error_Panel_4;
   #Enable_Comunication_Erro_7 := NOT #Comunication_Error_Panel_1 AND NOT #Comunication_Error_Panel_3 AND NOT #Comunication_Error_Panel_5;
   #Enable_Comunication_Erro_8 := NOT #Comunication_Error_Panel_2 AND NOT #Comunication_Error_Panel_4 AND NOT #Comunication_Error_Panel_6;
   #Enable_Comunication_Erro_9 := NOT #Comunication_Error_Panel_1 AND NOT #Comunication_Error_Panel_3 AND NOT #Comunication_Error_Panel_5 AND NOT #Comunication_Error_Panel_7;
   #Enable_Comunication_Erro_10 := NOT #Comunication_Error_Panel_2 AND NOT #Comunication_Error_Panel_4 AND NOT #Comunication_Error_Panel_6 AND NOT #Comunication_Error_Panel_8;
   #Enable_Comunication_Erro_11 := NOT #Comunication_Error_Panel_1 AND NOT #Comunication_Error_Panel_3 AND NOT #Comunication_Error_Panel_5 AND NOT #Comunication_Error_Panel_7 AND NOT #Comunication_Error_Panel_9;
   #Enable_Comunication_Erro_12 := NOT #Comunication_Error_Panel_2 AND NOT #Comunication_Error_Panel_4 AND NOT #Comunication_Error_Panel_6 AND NOT #Comunication_Error_Panel_8 AND NOT #Comunication_Error_Panel_10;
   #Enable_Comunication_Erro_13 := NOT #Comunication_Error_Panel_1 AND NOT #Comunication_Error_Panel_3 AND NOT #Comunication_Error_Panel_5 AND NOT #Comunication_Error_Panel_7 AND NOT #Comunication_Error_Panel_9 AND NOT #Comunication_Error_Panel_11;
   #Enable_Comunication_Erro_14 := NOT #Comunication_Error_Panel_2 AND NOT #Comunication_Error_Panel_4 AND NOT #Comunication_Error_Panel_6 AND NOT #Comunication_Error_Panel_8 AND NOT #Comunication_Error_Panel_10 AND NOT #Comunication_Error_Panel_12;
   #Enable_Comunication_Erro_15 := NOT #Comunication_Error_Panel_1 AND NOT #Comunication_Error_Panel_3 AND NOT #Comunication_Error_Panel_5 AND NOT #Comunication_Error_Panel_7 AND NOT #Comunication_Error_Panel_9 AND NOT #Comunication_Error_Panel_11 AND NOT #Comunication_Error_Panel_13;
   #Enable_Comunication_Erro_16 := NOT #Comunication_Error_Panel_2 AND NOT #Comunication_Error_Panel_4 AND NOT #Comunication_Error_Panel_6 AND NOT #Comunication_Error_Panel_8 AND NOT #Comunication_Error_Panel_10 AND NOT #Comunication_Error_Panel_12 AND NOT #Comunication_Error_Panel_14;
   #Enable_Comunication_Erro_17 := NOT #Comunication_Error_Panel_1 AND NOT #Comunication_Error_Panel_3 AND NOT #Comunication_Error_Panel_5 AND NOT #Comunication_Error_Panel_7 AND NOT #Comunication_Error_Panel_9 AND NOT #Comunication_Error_Panel_11 AND NOT #Comunication_Error_Panel_13 AND NOT #Comunication_Error_Panel_15;
   #Enable_Comunication_Erro_18 := NOT #Comunication_Error_Panel_2 AND NOT #Comunication_Error_Panel_4 AND NOT #Comunication_Error_Panel_6 AND NOT #Comunication_Error_Panel_8 AND NOT #Comunication_Error_Panel_10 AND NOT #Comunication_Error_Panel_12 AND NOT #Comunication_Error_Panel_14 AND NOT #Comunication_Error_Panel_16;
   #Enable_Comunication_Erro_19 := NOT #Comunication_Error_Panel_1 AND NOT #Comunication_Error_Panel_3 AND NOT #Comunication_Error_Panel_5 AND NOT #Comunication_Error_Panel_7 AND NOT #Comunication_Error_Panel_9 AND NOT #Comunication_Error_Panel_11 AND NOT #Comunication_Error_Panel_13 AND NOT #Comunication_Error_Panel_15 AND NOT #Comunication_Error_Panel_17;
   #Enable_Comunication_Erro_20 := NOT #Comunication_Error_Panel_2 AND NOT #Comunication_Error_Panel_4 AND NOT #Comunication_Error_Panel_6 AND NOT #Comunication_Error_Panel_8 AND NOT #Comunication_Error_Panel_10 AND NOT #Comunication_Error_Panel_12 AND NOT #Comunication_Error_Panel_14 AND NOT #Comunication_Error_Panel_16 AND NOT #Comunication_Error_Panel_18;
   #Enable_Comunication_Erro_21 := NOT #Comunication_Error_Panel_1 AND NOT #Comunication_Error_Panel_3 AND NOT #Comunication_Error_Panel_5 AND NOT #Comunication_Error_Panel_7 AND NOT #Comunication_Error_Panel_9 AND NOT #Comunication_Error_Panel_11 AND NOT #Comunication_Error_Panel_13 AND NOT #Comunication_Error_Panel_15 AND NOT #Comunication_Error_Panel_17 AND NOT #Comunication_Error_Panel_19;
   #Enable_Comunication_Erro_22 := NOT #Comunication_Error_Panel_2 AND NOT #Comunication_Error_Panel_4 AND NOT #Comunication_Error_Panel_6 AND NOT #Comunication_Error_Panel_8 AND NOT #Comunication_Error_Panel_10 AND NOT #Comunication_Error_Panel_12 AND NOT #Comunication_Error_Panel_14 AND NOT #Comunication_Error_Panel_16 AND NOT #Comunication_Error_Panel_18 AND NOT #Comunication_Error_Panel_20;
   #Enable_Comunication_Erro_23 := NOT #Comunication_Error_Panel_1 AND NOT #Comunication_Error_Panel_3 AND NOT #Comunication_Error_Panel_5 AND NOT #Comunication_Error_Panel_7 AND NOT #Comunication_Error_Panel_9 AND NOT #Comunication_Error_Panel_11 AND NOT #Comunication_Error_Panel_13 AND NOT #Comunication_Error_Panel_15 AND NOT #Comunication_Error_Panel_17 AND NOT #Comunication_Error_Panel_19 AND NOT #Comunication_Error_Panel_21;
   #Enable_Comunication_Erro_24 := NOT #Comunication_Error_Panel_2 AND NOT #Comunication_Error_Panel_4 AND NOT #Comunication_Error_Panel_6 AND NOT #Comunication_Error_Panel_8 AND NOT #Comunication_Error_Panel_10 AND NOT #Comunication_Error_Panel_12 AND NOT #Comunication_Error_Panel_14 AND NOT #Comunication_Error_Panel_16 AND NOT #Comunication_Error_Panel_18 AND NOT #Comunication_Error_Panel_20 AND NOT #Comunication_Error_Panel_22;
   #Enable_Comunication_Erro_25 := NOT #Comunication_Error_Panel_1 AND NOT #Comunication_Error_Panel_3 AND NOT #Comunication_Error_Panel_5 AND NOT #Comunication_Error_Panel_7 AND NOT #Comunication_Error_Panel_9 AND NOT #Comunication_Error_Panel_11 AND NOT #Comunication_Error_Panel_13 AND NOT #Comunication_Error_Panel_15 AND NOT #Comunication_Error_Panel_17 AND NOT #Comunication_Error_Panel_19 AND NOT #Comunication_Error_Panel_21 AND NOT #Comunication_Error_Panel_23;
   #Enable_Comunication_Erro_26 := NOT #Comunication_Error_Panel_2 AND NOT #Comunication_Error_Panel_4 AND NOT #Comunication_Error_Panel_6 AND NOT #Comunication_Error_Panel_8 AND NOT #Comunication_Error_Panel_10 AND NOT #Comunication_Error_Panel_12 AND NOT #Comunication_Error_Panel_14 AND NOT #Comunication_Error_Panel_16 AND NOT #Comunication_Error_Panel_18 AND NOT #Comunication_Error_Panel_20 AND NOT #Comunication_Error_Panel_22 AND NOT #Comunication_Error_Panel_24;
   #Enable_Comunication_Erro_27 := NOT #Comunication_Error_Panel_1 AND NOT #Comunication_Error_Panel_3 AND NOT #Comunication_Error_Panel_5 AND NOT #Comunication_Error_Panel_7 AND NOT #Comunication_Error_Panel_9 AND NOT #Comunication_Error_Panel_11 AND NOT #Comunication_Error_Panel_13 AND NOT #Comunication_Error_Panel_15 AND NOT #Comunication_Error_Panel_17 AND NOT #Comunication_Error_Panel_19 AND NOT #Comunication_Error_Panel_21 AND NOT #Comunication_Error_Panel_23 AND NOT #Comunication_Error_Panel_25;
   #Enable_Comunication_Erro_28 := NOT #Comunication_Error_Panel_2 AND NOT #Comunication_Error_Panel_4 AND NOT #Comunication_Error_Panel_6 AND NOT #Comunication_Error_Panel_8 AND NOT #Comunication_Error_Panel_10 AND NOT #Comunication_Error_Panel_12 AND NOT #Comunication_Error_Panel_14 AND NOT #Comunication_Error_Panel_16 AND NOT #Comunication_Error_Panel_18 AND NOT #Comunication_Error_Panel_20 AND NOT #Comunication_Error_Panel_22 AND NOT #Comunication_Error_Panel_24 AND NOT #Comunication_Error_Panel_26;
   #Enable_Comunication_Erro_29 := NOT #Comunication_Error_Panel_1 AND NOT #Comunication_Error_Panel_3 AND NOT #Comunication_Error_Panel_5 AND NOT #Comunication_Error_Panel_7 AND NOT #Comunication_Error_Panel_9 AND NOT #Comunication_Error_Panel_11 AND NOT #Comunication_Error_Panel_13 AND NOT #Comunication_Error_Panel_15 AND NOT #Comunication_Error_Panel_17 AND NOT #Comunication_Error_Panel_19 AND NOT #Comunication_Error_Panel_21 AND NOT #Comunication_Error_Panel_23 AND NOT #Comunication_Error_Panel_25 AND NOT #Comunication_Error_Panel_27;
   #Enable_Comunication_Erro_30 := NOT #Comunication_Error_Panel_2 AND NOT #Comunication_Error_Panel_4 AND NOT #Comunication_Error_Panel_6 AND NOT #Comunication_Error_Panel_8 AND NOT #Comunication_Error_Panel_10 AND NOT #Comunication_Error_Panel_12 AND NOT #Comunication_Error_Panel_14 AND NOT #Comunication_Error_Panel_16 AND NOT #Comunication_Error_Panel_18 AND NOT #Comunication_Error_Panel_20 AND NOT #Comunication_Error_Panel_22 AND NOT #Comunication_Error_Panel_24 AND NOT #Comunication_Error_Panel_26 AND NOT #Comunication_Error_Panel_28;
END_REGION

REGION Network 7
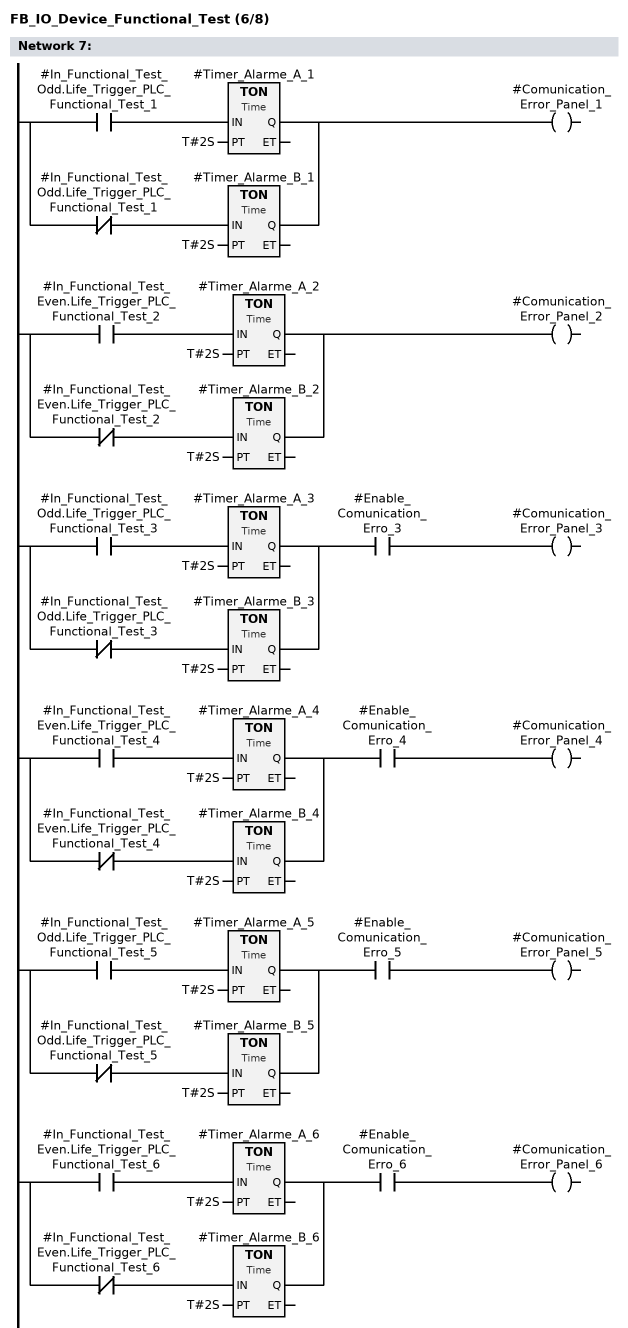
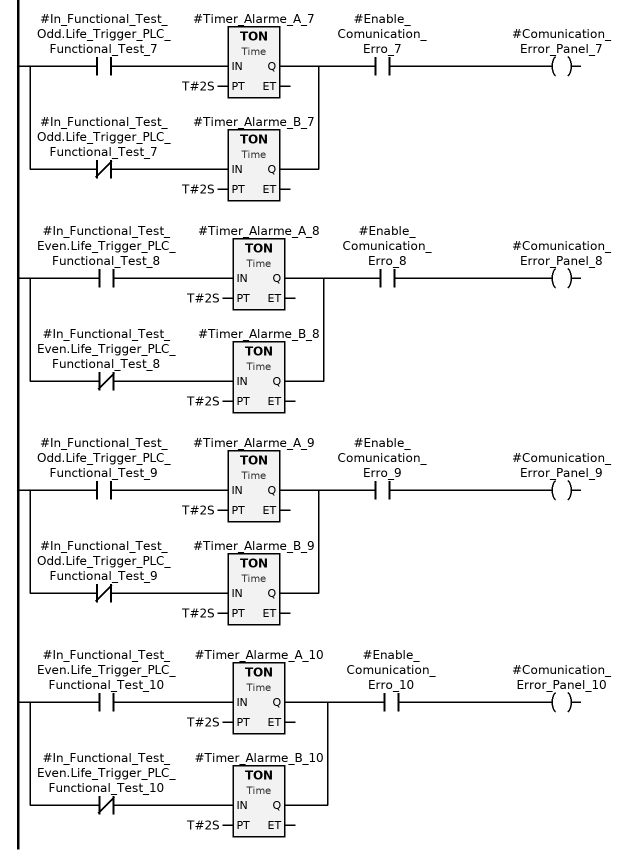
   RUNG wire#powerrail
      Contact( #In_Functional_Test_Odd.Life_Trigger_PLC_Functional_Test_1 )
      { S7_Templates := "time_type := Time" } #Timer_Alarme_A_1.TON(pt := T#2S, et =>)
      wire#w1
      Coil( #Comunication_Error_Panel_1 )
   END_RUNG
   RUNG wire#powerrail
      I_Contact( #In_Functional_Test_Odd.Life_Trigger_PLC_Functional_Test_1 )
      { S7_Templates := "time_type := Time" } #Timer_Alarme_B_1.TON(pt := T#2S, et =>)
   END_RUNG wire#w1
   RUNG wire#powerrail
      Contact( #In_Functional_Test_Even.Life_Trigger_PLC_Functional_Test_2 )
      { S7_Templates := "time_type := Time" } #Timer_Alarme_A_2.TON(pt := T#2S, et =>)
      wire#w2
      Coil( #Comunication_Error_Panel_2 )
   END_RUNG
   RUNG wire#powerrail
      I_Contact( #In_Functional_Test_Even.Life_Trigger_PLC_Functional_Test_2 )
      { S7_Templates := "time_type := Time" } #Timer_Alarme_B_2.TON(pt := T#2S, et =>)
   END_RUNG wire#w2
   RUNG wire#powerrail
      Contact( #In_Functional_Test_Odd.Life_Trigger_PLC_Functional_Test_3 )
      { S7_Templates := "time_type := Time" } #Timer_Alarme_A_3.TON(pt := T#2S, et =>)
      wire#w3
      Contact( #Enable_Comunication_Erro_3 )
      Coil( #Comunication_Error_Panel_3 )
   END_RUNG
   RUNG wire#powerrail
      I_Contact( #In_Functional_Test_Odd.Life_Trigger_PLC_Functional_Test_3 )
      { S7_Templates := "time_type := Time" } #Timer_Alarme_B_3.TON(pt := T#2S, et =>)
   END_RUNG wire#w3
   RUNG wire#powerrail
      Contact( #In_Functional_Test_Even.Life_Trigger_PLC_Functional_Test_4 )
      { S7_Templates := "time_type := Time" } #Timer_Alarme_A_4.TON(pt := T#2S, et =>)
      wire#w4
      Contact( #Enable_Comunication_Erro_4 )
      Coil( #Comunication_Error_Panel_4 )
   END_RUNG
   RUNG wire#powerrail
      I_Contact( #In_Functional_Test_Even.Life_Trigger_PLC_Functional_Test_4 )
      { S7_Templates := "time_type := Time" } #Timer_Alarme_B_4.TON(pt := T#2S, et =>)
   END_RUNG wire#w4
   RUNG wire#powerrail
      Contact( #In_Functional_Test_Odd.Life_Trigger_PLC_Functional_Test_5 )
      { S7_Templates := "time_type := Time" } #Timer_Alarme_A_5.TON(pt := T#2S, et =>)
      wire#w5
      Contact( #Enable_Comunication_Erro_5 )
      Coil( #Comunication_Error_Panel_5 )
   END_RUNG
   RUNG wire#powerrail
      I_Contact( #In_Functional_Test_Odd.Life_Trigger_PLC_Functional_Test_5 )
      { S7_Templates := "time_type := Time" } #Timer_Alarme_B_5.TON(pt := T#2S, et =>)
   END_RUNG wire#w5
   RUNG wire#powerrail
      Contact( #In_Functional_Test_Even.Life_Trigger_PLC_Functional_Test_6 )
      { S7_Templates := "time_type := Time" } #Timer_Alarme_A_6.TON(pt := T#2S, et =>)
      wire#w6
      Contact( #Enable_Comunication_Erro_6 )
      Coil( #Comunication_Error_Panel_6 )
   END_RUNG
   RUNG wire#powerrail
      I_Contact( #In_Functional_Test_Even.Life_Trigger_PLC_Functional_Test_6 )
      { S7_Templates := "time_type := Time" } #Timer_Alarme_B_6.TON(pt := T#2S, et =>)
   END_RUNG wire#w6
   RUNG wire#powerrail
      Contact( #In_Functional_Test_Odd.Life_Trigger_PLC_Functional_Test_7 )
      { S7_Templates := "time_type := Time" } #Timer_Alarme_A_7.TON(pt := T#2S, et =>)
      wire#w7
      Contact( #Enable_Comunication_Erro_7 )
      Coil( #Comunication_Error_Panel_7 )
   END_RUNG
   RUNG wire#powerrail
      I_Contact( #In_Functional_Test_Odd.Life_Trigger_PLC_Functional_Test_7 )
      { S7_Templates := "time_type := Time" } #Timer_Alarme_B_7.TON(pt := T#2S, et =>)
   END_RUNG wire#w7
   RUNG wire#powerrail
      Contact( #In_Functional_Test_Even.Life_Trigger_PLC_Functional_Test_8 )
      { S7_Templates := "time_type := Time" } #Timer_Alarme_A_8.TON(pt := T#2S, et =>)
      wire#w8
      Contact( #Enable_Comunication_Erro_8 )
      Coil( #Comunication_Error_Panel_8 )
   END_RUNG
   RUNG wire#powerrail
      I_Contact( #In_Functional_Test_Even.Life_Trigger_PLC_Functional_Test_8 )
      { S7_Templates := "time_type := Time" } #Timer_Alarme_B_8.TON(pt := T#2S, et =>)
   END_RUNG wire#w8
   RUNG wire#powerrail
      Contact( #In_Functional_Test_Odd.Life_Trigger_PLC_Functional_Test_9 )
      { S7_Templates := "time_type := Time" } #Timer_Alarme_A_9.TON(pt := T#2S, et =>)
      wire#w9
      Contact( #Enable_Comunication_Erro_9 )
      Coil( #Comunication_Error_Panel_9 )
   END_RUNG
   RUNG wire#powerrail
      I_Contact( #In_Functional_Test_Odd.Life_Trigger_PLC_Functional_Test_9 )
      { S7_Templates := "time_type := Time" } #Timer_Alarme_B_9.TON(pt := T#2S, et =>)
   END_RUNG wire#w9
   RUNG wire#powerrail
      Contact( #In_Functional_Test_Even.Life_Trigger_PLC_Functional_Test_10 )
      { S7_Templates := "time_type := Time" } #Timer_Alarme_A_10.TON(pt := T#2S, et =>)
      wire#w10
      Contact( #Enable_Comunication_Erro_10 )
      Coil( #Comunication_Error_Panel_10 )
   END_RUNG
   RUNG wire#powerrail
      I_Contact( #In_Functional_Test_Even.Life_Trigger_PLC_Functional_Test_10 )
      { S7_Templates := "time_type := Time" } #Timer_Alarme_B_10.TON(pt := T#2S, et =>)
   END_RUNG wire#w10
   // the same network as SCL:
   #Timer_Alarme_A_1(IN := #In_Functional_Test_Odd.Life_Trigger_PLC_Functional_Test_1, PT := T#2S);   // TON
   #Timer_Alarme_B_1(IN := NOT #In_Functional_Test_Odd.Life_Trigger_PLC_Functional_Test_1, PT := T#2S);   // TON
   #Comunication_Error_Panel_1 := #Timer_Alarme_A_1.Q OR #Timer_Alarme_B_1.Q;
   #Timer_Alarme_A_2(IN := #In_Functional_Test_Even.Life_Trigger_PLC_Functional_Test_2, PT := T#2S);   // TON
   #Timer_Alarme_B_2(IN := NOT #In_Functional_Test_Even.Life_Trigger_PLC_Functional_Test_2, PT := T#2S);   // TON
   #Comunication_Error_Panel_2 := #Timer_Alarme_A_2.Q OR #Timer_Alarme_B_2.Q;
   #Timer_Alarme_A_3(IN := #In_Functional_Test_Odd.Life_Trigger_PLC_Functional_Test_3, PT := T#2S);   // TON
   #Timer_Alarme_B_3(IN := NOT #In_Functional_Test_Odd.Life_Trigger_PLC_Functional_Test_3, PT := T#2S);   // TON
   #Comunication_Error_Panel_3 := (#Timer_Alarme_A_3.Q OR #Timer_Alarme_B_3.Q) AND #Enable_Comunication_Erro_3;
   #Timer_Alarme_A_4(IN := #In_Functional_Test_Even.Life_Trigger_PLC_Functional_Test_4, PT := T#2S);   // TON
   #Timer_Alarme_B_4(IN := NOT #In_Functional_Test_Even.Life_Trigger_PLC_Functional_Test_4, PT := T#2S);   // TON
   #Comunication_Error_Panel_4 := (#Timer_Alarme_A_4.Q OR #Timer_Alarme_B_4.Q) AND #Enable_Comunication_Erro_4;
   #Timer_Alarme_A_5(IN := #In_Functional_Test_Odd.Life_Trigger_PLC_Functional_Test_5, PT := T#2S);   // TON
   #Timer_Alarme_B_5(IN := NOT #In_Functional_Test_Odd.Life_Trigger_PLC_Functional_Test_5, PT := T#2S);   // TON
   #Comunication_Error_Panel_5 := (#Timer_Alarme_A_5.Q OR #Timer_Alarme_B_5.Q) AND #Enable_Comunication_Erro_5;
   #Timer_Alarme_A_6(IN := #In_Functional_Test_Even.Life_Trigger_PLC_Functional_Test_6, PT := T#2S);   // TON
   #Timer_Alarme_B_6(IN := NOT #In_Functional_Test_Even.Life_Trigger_PLC_Functional_Test_6, PT := T#2S);   // TON
   #Comunication_Error_Panel_6 := (#Timer_Alarme_A_6.Q OR #Timer_Alarme_B_6.Q) AND #Enable_Comunication_Erro_6;
   #Timer_Alarme_A_7(IN := #In_Functional_Test_Odd.Life_Trigger_PLC_Functional_Test_7, PT := T#2S);   // TON
   #Timer_Alarme_B_7(IN := NOT #In_Functional_Test_Odd.Life_Trigger_PLC_Functional_Test_7, PT := T#2S);   // TON
   #Comunication_Error_Panel_7 := (#Timer_Alarme_A_7.Q OR #Timer_Alarme_B_7.Q) AND #Enable_Comunication_Erro_7;
   #Timer_Alarme_A_8(IN := #In_Functional_Test_Even.Life_Trigger_PLC_Functional_Test_8, PT := T#2S);   // TON
   #Timer_Alarme_B_8(IN := NOT #In_Functional_Test_Even.Life_Trigger_PLC_Functional_Test_8, PT := T#2S);   // TON
   #Comunication_Error_Panel_8 := (#Timer_Alarme_A_8.Q OR #Timer_Alarme_B_8.Q) AND #Enable_Comunication_Erro_8;
   #Timer_Alarme_A_9(IN := #In_Functional_Test_Odd.Life_Trigger_PLC_Functional_Test_9, PT := T#2S);   // TON
   #Timer_Alarme_B_9(IN := NOT #In_Functional_Test_Odd.Life_Trigger_PLC_Functional_Test_9, PT := T#2S);   // TON
   #Comunication_Error_Panel_9 := (#Timer_Alarme_A_9.Q OR #Timer_Alarme_B_9.Q) AND #Enable_Comunication_Erro_9;
   #Timer_Alarme_A_10(IN := #In_Functional_Test_Even.Life_Trigger_PLC_Functional_Test_10, PT := T#2S);   // TON
   #Timer_Alarme_B_10(IN := NOT #In_Functional_Test_Even.Life_Trigger_PLC_Functional_Test_10, PT := T#2S);   // TON
   #Comunication_Error_Panel_10 := (#Timer_Alarme_A_10.Q OR #Timer_Alarme_B_10.Q) AND #Enable_Comunication_Erro_10;
END_REGION

REGION Network 8
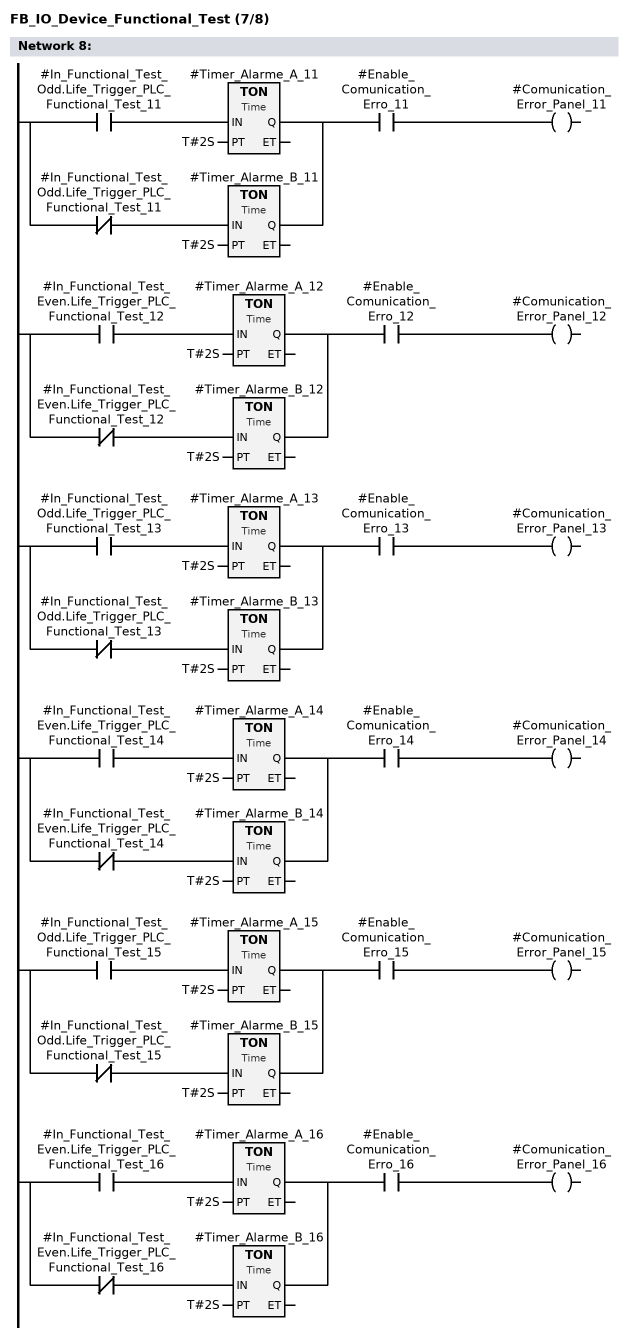
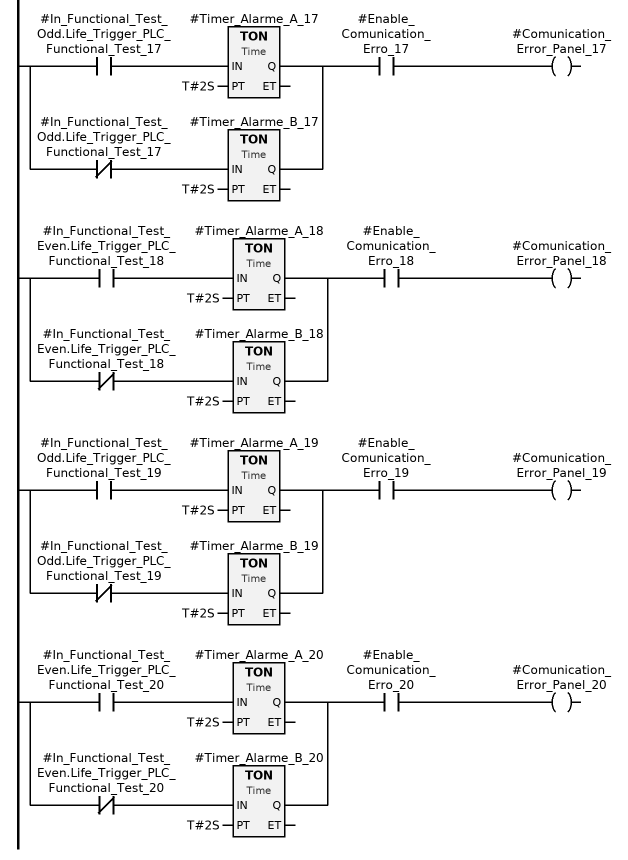
   RUNG wire#powerrail
      Contact( #In_Functional_Test_Odd.Life_Trigger_PLC_Functional_Test_11 )
      { S7_Templates := "time_type := Time" } #Timer_Alarme_A_11.TON(pt := T#2S, et =>)
      wire#w1
      Contact( #Enable_Comunication_Erro_11 )
      Coil( #Comunication_Error_Panel_11 )
   END_RUNG
   RUNG wire#powerrail
      I_Contact( #In_Functional_Test_Odd.Life_Trigger_PLC_Functional_Test_11 )
      { S7_Templates := "time_type := Time" } #Timer_Alarme_B_11.TON(pt := T#2S, et =>)
   END_RUNG wire#w1
   RUNG wire#powerrail
      Contact( #In_Functional_Test_Even.Life_Trigger_PLC_Functional_Test_12 )
      { S7_Templates := "time_type := Time" } #Timer_Alarme_A_12.TON(pt := T#2S, et =>)
      wire#w2
      Contact( #Enable_Comunication_Erro_12 )
      Coil( #Comunication_Error_Panel_12 )
   END_RUNG
   RUNG wire#powerrail
      I_Contact( #In_Functional_Test_Even.Life_Trigger_PLC_Functional_Test_12 )
      { S7_Templates := "time_type := Time" } #Timer_Alarme_B_12.TON(pt := T#2S, et =>)
   END_RUNG wire#w2
   RUNG wire#powerrail
      Contact( #In_Functional_Test_Odd.Life_Trigger_PLC_Functional_Test_13 )
      { S7_Templates := "time_type := Time" } #Timer_Alarme_A_13.TON(pt := T#2S, et =>)
      wire#w3
      Contact( #Enable_Comunication_Erro_13 )
      Coil( #Comunication_Error_Panel_13 )
   END_RUNG
   RUNG wire#powerrail
      I_Contact( #In_Functional_Test_Odd.Life_Trigger_PLC_Functional_Test_13 )
      { S7_Templates := "time_type := Time" } #Timer_Alarme_B_13.TON(pt := T#2S, et =>)
   END_RUNG wire#w3
   RUNG wire#powerrail
      Contact( #In_Functional_Test_Even.Life_Trigger_PLC_Functional_Test_14 )
      { S7_Templates := "time_type := Time" } #Timer_Alarme_A_14.TON(pt := T#2S, et =>)
      wire#w4
      Contact( #Enable_Comunication_Erro_14 )
      Coil( #Comunication_Error_Panel_14 )
   END_RUNG
   RUNG wire#powerrail
      I_Contact( #In_Functional_Test_Even.Life_Trigger_PLC_Functional_Test_14 )
      { S7_Templates := "time_type := Time" } #Timer_Alarme_B_14.TON(pt := T#2S, et =>)
   END_RUNG wire#w4
   RUNG wire#powerrail
      Contact( #In_Functional_Test_Odd.Life_Trigger_PLC_Functional_Test_15 )
      { S7_Templates := "time_type := Time" } #Timer_Alarme_A_15.TON(pt := T#2S, et =>)
      wire#w5
      Contact( #Enable_Comunication_Erro_15 )
      Coil( #Comunication_Error_Panel_15 )
   END_RUNG
   RUNG wire#powerrail
      I_Contact( #In_Functional_Test_Odd.Life_Trigger_PLC_Functional_Test_15 )
      { S7_Templates := "time_type := Time" } #Timer_Alarme_B_15.TON(pt := T#2S, et =>)
   END_RUNG wire#w5
   RUNG wire#powerrail
      Contact( #In_Functional_Test_Even.Life_Trigger_PLC_Functional_Test_16 )
      { S7_Templates := "time_type := Time" } #Timer_Alarme_A_16.TON(pt := T#2S, et =>)
      wire#w6
      Contact( #Enable_Comunication_Erro_16 )
      Coil( #Comunication_Error_Panel_16 )
   END_RUNG
   RUNG wire#powerrail
      I_Contact( #In_Functional_Test_Even.Life_Trigger_PLC_Functional_Test_16 )
      { S7_Templates := "time_type := Time" } #Timer_Alarme_B_16.TON(pt := T#2S, et =>)
   END_RUNG wire#w6
   RUNG wire#powerrail
      Contact( #In_Functional_Test_Odd.Life_Trigger_PLC_Functional_Test_17 )
      { S7_Templates := "time_type := Time" } #Timer_Alarme_A_17.TON(pt := T#2S, et =>)
      wire#w7
      Contact( #Enable_Comunication_Erro_17 )
      Coil( #Comunication_Error_Panel_17 )
   END_RUNG
   RUNG wire#powerrail
      I_Contact( #In_Functional_Test_Odd.Life_Trigger_PLC_Functional_Test_17 )
      { S7_Templates := "time_type := Time" } #Timer_Alarme_B_17.TON(pt := T#2S, et =>)
   END_RUNG wire#w7
   RUNG wire#powerrail
      Contact( #In_Functional_Test_Even.Life_Trigger_PLC_Functional_Test_18 )
      { S7_Templates := "time_type := Time" } #Timer_Alarme_A_18.TON(pt := T#2S, et =>)
      wire#w8
      Contact( #Enable_Comunication_Erro_18 )
      Coil( #Comunication_Error_Panel_18 )
   END_RUNG
   RUNG wire#powerrail
      I_Contact( #In_Functional_Test_Even.Life_Trigger_PLC_Functional_Test_18 )
      { S7_Templates := "time_type := Time" } #Timer_Alarme_B_18.TON(pt := T#2S, et =>)
   END_RUNG wire#w8
   RUNG wire#powerrail
      Contact( #In_Functional_Test_Odd.Life_Trigger_PLC_Functional_Test_19 )
      { S7_Templates := "time_type := Time" } #Timer_Alarme_A_19.TON(pt := T#2S, et =>)
      wire#w9
      Contact( #Enable_Comunication_Erro_19 )
      Coil( #Comunication_Error_Panel_19 )
   END_RUNG
   RUNG wire#powerrail
      I_Contact( #In_Functional_Test_Odd.Life_Trigger_PLC_Functional_Test_19 )
      { S7_Templates := "time_type := Time" } #Timer_Alarme_B_19.TON(pt := T#2S, et =>)
   END_RUNG wire#w9
   RUNG wire#powerrail
      Contact( #In_Functional_Test_Even.Life_Trigger_PLC_Functional_Test_20 )
      { S7_Templates := "time_type := Time" } #Timer_Alarme_A_20.TON(pt := T#2S, et =>)
      wire#w10
      Contact( #Enable_Comunication_Erro_20 )
      Coil( #Comunication_Error_Panel_20 )
   END_RUNG
   RUNG wire#powerrail
      I_Contact( #In_Functional_Test_Even.Life_Trigger_PLC_Functional_Test_20 )
      { S7_Templates := "time_type := Time" } #Timer_Alarme_B_20.TON(pt := T#2S, et =>)
   END_RUNG wire#w10
   // the same network as SCL:
   #Timer_Alarme_A_11(IN := #In_Functional_Test_Odd.Life_Trigger_PLC_Functional_Test_11, PT := T#2S);   // TON
   #Timer_Alarme_B_11(IN := NOT #In_Functional_Test_Odd.Life_Trigger_PLC_Functional_Test_11, PT := T#2S);   // TON
   #Comunication_Error_Panel_11 := (#Timer_Alarme_A_11.Q OR #Timer_Alarme_B_11.Q) AND #Enable_Comunication_Erro_11;
   #Timer_Alarme_A_12(IN := #In_Functional_Test_Even.Life_Trigger_PLC_Functional_Test_12, PT := T#2S);   // TON
   #Timer_Alarme_B_12(IN := NOT #In_Functional_Test_Even.Life_Trigger_PLC_Functional_Test_12, PT := T#2S);   // TON
   #Comunication_Error_Panel_12 := (#Timer_Alarme_A_12.Q OR #Timer_Alarme_B_12.Q) AND #Enable_Comunication_Erro_12;
   #Timer_Alarme_A_13(IN := #In_Functional_Test_Odd.Life_Trigger_PLC_Functional_Test_13, PT := T#2S);   // TON
   #Timer_Alarme_B_13(IN := NOT #In_Functional_Test_Odd.Life_Trigger_PLC_Functional_Test_13, PT := T#2S);   // TON
   #Comunication_Error_Panel_13 := (#Timer_Alarme_A_13.Q OR #Timer_Alarme_B_13.Q) AND #Enable_Comunication_Erro_13;
   #Timer_Alarme_A_14(IN := #In_Functional_Test_Even.Life_Trigger_PLC_Functional_Test_14, PT := T#2S);   // TON
   #Timer_Alarme_B_14(IN := NOT #In_Functional_Test_Even.Life_Trigger_PLC_Functional_Test_14, PT := T#2S);   // TON
   #Comunication_Error_Panel_14 := (#Timer_Alarme_A_14.Q OR #Timer_Alarme_B_14.Q) AND #Enable_Comunication_Erro_14;
   #Timer_Alarme_A_15(IN := #In_Functional_Test_Odd.Life_Trigger_PLC_Functional_Test_15, PT := T#2S);   // TON
   #Timer_Alarme_B_15(IN := NOT #In_Functional_Test_Odd.Life_Trigger_PLC_Functional_Test_15, PT := T#2S);   // TON
   #Comunication_Error_Panel_15 := (#Timer_Alarme_A_15.Q OR #Timer_Alarme_B_15.Q) AND #Enable_Comunication_Erro_15;
   #Timer_Alarme_A_16(IN := #In_Functional_Test_Even.Life_Trigger_PLC_Functional_Test_16, PT := T#2S);   // TON
   #Timer_Alarme_B_16(IN := NOT #In_Functional_Test_Even.Life_Trigger_PLC_Functional_Test_16, PT := T#2S);   // TON
   #Comunication_Error_Panel_16 := (#Timer_Alarme_A_16.Q OR #Timer_Alarme_B_16.Q) AND #Enable_Comunication_Erro_16;
   #Timer_Alarme_A_17(IN := #In_Functional_Test_Odd.Life_Trigger_PLC_Functional_Test_17, PT := T#2S);   // TON
   #Timer_Alarme_B_17(IN := NOT #In_Functional_Test_Odd.Life_Trigger_PLC_Functional_Test_17, PT := T#2S);   // TON
   #Comunication_Error_Panel_17 := (#Timer_Alarme_A_17.Q OR #Timer_Alarme_B_17.Q) AND #Enable_Comunication_Erro_17;
   #Timer_Alarme_A_18(IN := #In_Functional_Test_Even.Life_Trigger_PLC_Functional_Test_18, PT := T#2S);   // TON
   #Timer_Alarme_B_18(IN := NOT #In_Functional_Test_Even.Life_Trigger_PLC_Functional_Test_18, PT := T#2S);   // TON
   #Comunication_Error_Panel_18 := (#Timer_Alarme_A_18.Q OR #Timer_Alarme_B_18.Q) AND #Enable_Comunication_Erro_18;
   #Timer_Alarme_A_19(IN := #In_Functional_Test_Odd.Life_Trigger_PLC_Functional_Test_19, PT := T#2S);   // TON
   #Timer_Alarme_B_19(IN := NOT #In_Functional_Test_Odd.Life_Trigger_PLC_Functional_Test_19, PT := T#2S);   // TON
   #Comunication_Error_Panel_19 := (#Timer_Alarme_A_19.Q OR #Timer_Alarme_B_19.Q) AND #Enable_Comunication_Erro_19;
   #Timer_Alarme_A_20(IN := #In_Functional_Test_Even.Life_Trigger_PLC_Functional_Test_20, PT := T#2S);   // TON
   #Timer_Alarme_B_20(IN := NOT #In_Functional_Test_Even.Life_Trigger_PLC_Functional_Test_20, PT := T#2S);   // TON
   #Comunication_Error_Panel_20 := (#Timer_Alarme_A_20.Q OR #Timer_Alarme_B_20.Q) AND #Enable_Comunication_Erro_20;
END_REGION

REGION Network 9
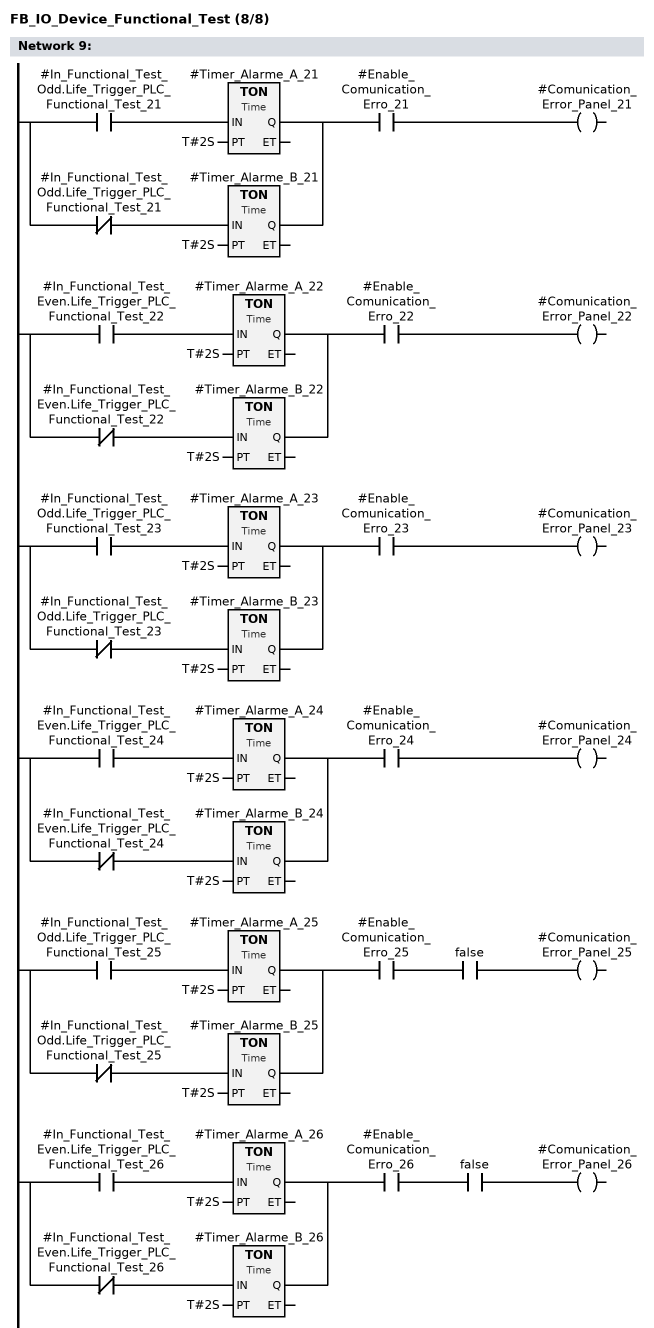
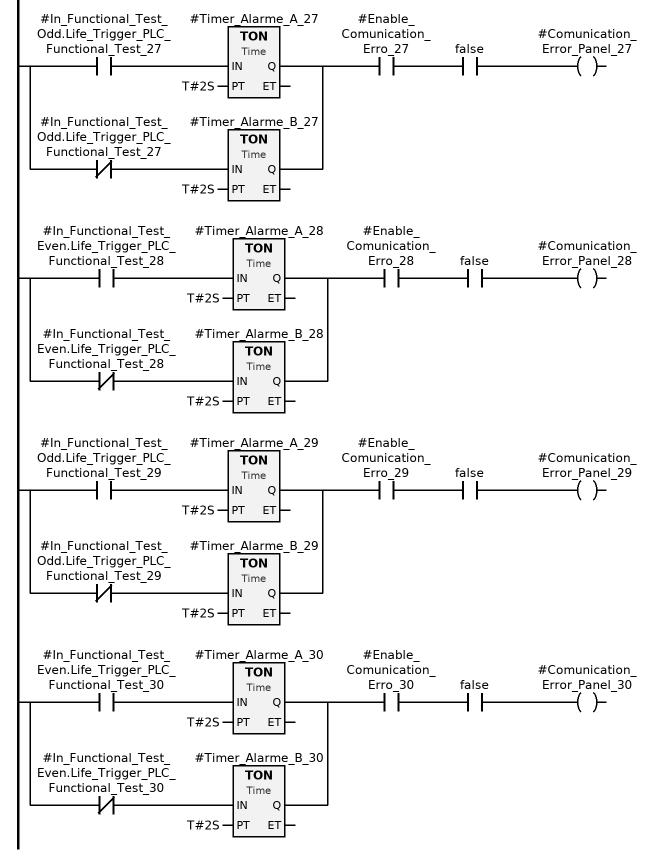
   RUNG wire#powerrail
      Contact( #In_Functional_Test_Odd.Life_Trigger_PLC_Functional_Test_21 )
      { S7_Templates := "time_type := Time" } #Timer_Alarme_A_21.TON(pt := T#2S, et =>)
      wire#w1
      Contact( #Enable_Comunication_Erro_21 )
      Coil( #Comunication_Error_Panel_21 )
   END_RUNG
   RUNG wire#powerrail
      I_Contact( #In_Functional_Test_Odd.Life_Trigger_PLC_Functional_Test_21 )
      { S7_Templates := "time_type := Time" } #Timer_Alarme_B_21.TON(pt := T#2S, et =>)
   END_RUNG wire#w1
   RUNG wire#powerrail
      Contact( #In_Functional_Test_Even.Life_Trigger_PLC_Functional_Test_22 )
      { S7_Templates := "time_type := Time" } #Timer_Alarme_A_22.TON(pt := T#2S, et =>)
      wire#w2
      Contact( #Enable_Comunication_Erro_22 )
      Coil( #Comunication_Error_Panel_22 )
   END_RUNG
   RUNG wire#powerrail
      I_Contact( #In_Functional_Test_Even.Life_Trigger_PLC_Functional_Test_22 )
      { S7_Templates := "time_type := Time" } #Timer_Alarme_B_22.TON(pt := T#2S, et =>)
   END_RUNG wire#w2
   RUNG wire#powerrail
      Contact( #In_Functional_Test_Odd.Life_Trigger_PLC_Functional_Test_23 )
      { S7_Templates := "time_type := Time" } #Timer_Alarme_A_23.TON(pt := T#2S, et =>)
      wire#w3
      Contact( #Enable_Comunication_Erro_23 )
      Coil( #Comunication_Error_Panel_23 )
   END_RUNG
   RUNG wire#powerrail
      I_Contact( #In_Functional_Test_Odd.Life_Trigger_PLC_Functional_Test_23 )
      { S7_Templates := "time_type := Time" } #Timer_Alarme_B_23.TON(pt := T#2S, et =>)
   END_RUNG wire#w3
   RUNG wire#powerrail
      Contact( #In_Functional_Test_Even.Life_Trigger_PLC_Functional_Test_24 )
      { S7_Templates := "time_type := Time" } #Timer_Alarme_A_24.TON(pt := T#2S, et =>)
      wire#w4
      Contact( #Enable_Comunication_Erro_24 )
      Coil( #Comunication_Error_Panel_24 )
   END_RUNG
   RUNG wire#powerrail
      I_Contact( #In_Functional_Test_Even.Life_Trigger_PLC_Functional_Test_24 )
      { S7_Templates := "time_type := Time" } #Timer_Alarme_B_24.TON(pt := T#2S, et =>)
   END_RUNG wire#w4
   RUNG wire#powerrail
      Contact( #In_Functional_Test_Odd.Life_Trigger_PLC_Functional_Test_25 )
      { S7_Templates := "time_type := Time" } #Timer_Alarme_A_25.TON(pt := T#2S, et =>)
      wire#w5
      Contact( #Enable_Comunication_Erro_25 )
      Contact( false )
      Coil( #Comunication_Error_Panel_25 )
   END_RUNG
   RUNG wire#powerrail
      I_Contact( #In_Functional_Test_Odd.Life_Trigger_PLC_Functional_Test_25 )
      { S7_Templates := "time_type := Time" } #Timer_Alarme_B_25.TON(pt := T#2S, et =>)
   END_RUNG wire#w5
   RUNG wire#powerrail
      Contact( #In_Functional_Test_Even.Life_Trigger_PLC_Functional_Test_26 )
      { S7_Templates := "time_type := Time" } #Timer_Alarme_A_26.TON(pt := T#2S, et =>)
      wire#w6
      Contact( #Enable_Comunication_Erro_26 )
      Contact( false )
      Coil( #Comunication_Error_Panel_26 )
   END_RUNG
   RUNG wire#powerrail
      I_Contact( #In_Functional_Test_Even.Life_Trigger_PLC_Functional_Test_26 )
      { S7_Templates := "time_type := Time" } #Timer_Alarme_B_26.TON(pt := T#2S, et =>)
   END_RUNG wire#w6
   RUNG wire#powerrail
      Contact( #In_Functional_Test_Odd.Life_Trigger_PLC_Functional_Test_27 )
      { S7_Templates := "time_type := Time" } #Timer_Alarme_A_27.TON(pt := T#2S, et =>)
      wire#w7
      Contact( #Enable_Comunication_Erro_27 )
      Contact( false )
      Coil( #Comunication_Error_Panel_27 )
   END_RUNG
   RUNG wire#powerrail
      I_Contact( #In_Functional_Test_Odd.Life_Trigger_PLC_Functional_Test_27 )
      { S7_Templates := "time_type := Time" } #Timer_Alarme_B_27.TON(pt := T#2S, et =>)
   END_RUNG wire#w7
   RUNG wire#powerrail
      Contact( #In_Functional_Test_Even.Life_Trigger_PLC_Functional_Test_28 )
      { S7_Templates := "time_type := Time" } #Timer_Alarme_A_28.TON(pt := T#2S, et =>)
      wire#w8
      Contact( #Enable_Comunication_Erro_28 )
      Contact( false )
      Coil( #Comunication_Error_Panel_28 )
   END_RUNG
   RUNG wire#powerrail
      I_Contact( #In_Functional_Test_Even.Life_Trigger_PLC_Functional_Test_28 )
      { S7_Templates := "time_type := Time" } #Timer_Alarme_B_28.TON(pt := T#2S, et =>)
   END_RUNG wire#w8
   RUNG wire#powerrail
      Contact( #In_Functional_Test_Odd.Life_Trigger_PLC_Functional_Test_29 )
      { S7_Templates := "time_type := Time" } #Timer_Alarme_A_29.TON(pt := T#2S, et =>)
      wire#w9
      Contact( #Enable_Comunication_Erro_29 )
      Contact( false )
      Coil( #Comunication_Error_Panel_29 )
   END_RUNG
   RUNG wire#powerrail
      I_Contact( #In_Functional_Test_Odd.Life_Trigger_PLC_Functional_Test_29 )
      { S7_Templates := "time_type := Time" } #Timer_Alarme_B_29.TON(pt := T#2S, et =>)
   END_RUNG wire#w9
   RUNG wire#powerrail
      Contact( #In_Functional_Test_Even.Life_Trigger_PLC_Functional_Test_30 )
      { S7_Templates := "time_type := Time" } #Timer_Alarme_A_30.TON(pt := T#2S, et =>)
      wire#w10
      Contact( #Enable_Comunication_Erro_30 )
      Contact( false )
      Coil( #Comunication_Error_Panel_30 )
   END_RUNG
   RUNG wire#powerrail
      I_Contact( #In_Functional_Test_Even.Life_Trigger_PLC_Functional_Test_30 )
      { S7_Templates := "time_type := Time" } #Timer_Alarme_B_30.TON(pt := T#2S, et =>)
   END_RUNG wire#w10
   // the same network as SCL:
   #Timer_Alarme_A_21(IN := #In_Functional_Test_Odd.Life_Trigger_PLC_Functional_Test_21, PT := T#2S);   // TON
   #Timer_Alarme_B_21(IN := NOT #In_Functional_Test_Odd.Life_Trigger_PLC_Functional_Test_21, PT := T#2S);   // TON
   #Comunication_Error_Panel_21 := (#Timer_Alarme_A_21.Q OR #Timer_Alarme_B_21.Q) AND #Enable_Comunication_Erro_21;
   #Timer_Alarme_A_22(IN := #In_Functional_Test_Even.Life_Trigger_PLC_Functional_Test_22, PT := T#2S);   // TON
   #Timer_Alarme_B_22(IN := NOT #In_Functional_Test_Even.Life_Trigger_PLC_Functional_Test_22, PT := T#2S);   // TON
   #Comunication_Error_Panel_22 := (#Timer_Alarme_A_22.Q OR #Timer_Alarme_B_22.Q) AND #Enable_Comunication_Erro_22;
   #Timer_Alarme_A_23(IN := #In_Functional_Test_Odd.Life_Trigger_PLC_Functional_Test_23, PT := T#2S);   // TON
   #Timer_Alarme_B_23(IN := NOT #In_Functional_Test_Odd.Life_Trigger_PLC_Functional_Test_23, PT := T#2S);   // TON
   #Comunication_Error_Panel_23 := (#Timer_Alarme_A_23.Q OR #Timer_Alarme_B_23.Q) AND #Enable_Comunication_Erro_23;
   #Timer_Alarme_A_24(IN := #In_Functional_Test_Even.Life_Trigger_PLC_Functional_Test_24, PT := T#2S);   // TON
   #Timer_Alarme_B_24(IN := NOT #In_Functional_Test_Even.Life_Trigger_PLC_Functional_Test_24, PT := T#2S);   // TON
   #Comunication_Error_Panel_24 := (#Timer_Alarme_A_24.Q OR #Timer_Alarme_B_24.Q) AND #Enable_Comunication_Erro_24;
   #Timer_Alarme_A_25(IN := #In_Functional_Test_Odd.Life_Trigger_PLC_Functional_Test_25, PT := T#2S);   // TON
   #Timer_Alarme_B_25(IN := NOT #In_Functional_Test_Odd.Life_Trigger_PLC_Functional_Test_25, PT := T#2S);   // TON
   #Comunication_Error_Panel_25 := (#Timer_Alarme_A_25.Q OR #Timer_Alarme_B_25.Q) AND #Enable_Comunication_Erro_25 AND false;
   #Timer_Alarme_A_26(IN := #In_Functional_Test_Even.Life_Trigger_PLC_Functional_Test_26, PT := T#2S);   // TON
   #Timer_Alarme_B_26(IN := NOT #In_Functional_Test_Even.Life_Trigger_PLC_Functional_Test_26, PT := T#2S);   // TON
   #Comunication_Error_Panel_26 := (#Timer_Alarme_A_26.Q OR #Timer_Alarme_B_26.Q) AND #Enable_Comunication_Erro_26 AND false;
   #Timer_Alarme_A_27(IN := #In_Functional_Test_Odd.Life_Trigger_PLC_Functional_Test_27, PT := T#2S);   // TON
   #Timer_Alarme_B_27(IN := NOT #In_Functional_Test_Odd.Life_Trigger_PLC_Functional_Test_27, PT := T#2S);   // TON
   #Comunication_Error_Panel_27 := (#Timer_Alarme_A_27.Q OR #Timer_Alarme_B_27.Q) AND #Enable_Comunication_Erro_27 AND false;
   #Timer_Alarme_A_28(IN := #In_Functional_Test_Even.Life_Trigger_PLC_Functional_Test_28, PT := T#2S);   // TON
   #Timer_Alarme_B_28(IN := NOT #In_Functional_Test_Even.Life_Trigger_PLC_Functional_Test_28, PT := T#2S);   // TON
   #Comunication_Error_Panel_28 := (#Timer_Alarme_A_28.Q OR #Timer_Alarme_B_28.Q) AND #Enable_Comunication_Erro_28 AND false;
   #Timer_Alarme_A_29(IN := #In_Functional_Test_Odd.Life_Trigger_PLC_Functional_Test_29, PT := T#2S);   // TON
   #Timer_Alarme_B_29(IN := NOT #In_Functional_Test_Odd.Life_Trigger_PLC_Functional_Test_29, PT := T#2S);   // TON
   #Comunication_Error_Panel_29 := (#Timer_Alarme_A_29.Q OR #Timer_Alarme_B_29.Q) AND #Enable_Comunication_Erro_29 AND false;
   #Timer_Alarme_A_30(IN := #In_Functional_Test_Even.Life_Trigger_PLC_Functional_Test_30, PT := T#2S);   // TON
   #Timer_Alarme_B_30(IN := NOT #In_Functional_Test_Even.Life_Trigger_PLC_Functional_Test_30, PT := T#2S);   // TON
   #Comunication_Error_Panel_30 := (#Timer_Alarme_A_30.Q OR #Timer_Alarme_B_30.Q) AND #Enable_Comunication_Erro_30 AND false;
END_REGION
END_FUNCTION_BLOCK
